DATA_BLOCK "NC"	// DB 10
VERSION : 0.0
  STRUCT
   A_Disabl_Inp1 : BOOL ;	//Disable digi. NCK input 1
   A_Disabl_Inp2 : BOOL ;	//Disable digi. NCK input 2
   A_Disabl_Inp3 : BOOL ;	//Disable digi. NCK input 3
   A_Disabl_Inp4 : BOOL ;	//Disable digi. NCK input 4
   A_Disabl_Inp5 : BOOL ;	//Disable digi. NCK input 5
   A_Disabl_Inp6 : BOOL ;	//Disable digi. NCK input 6
   A_Disabl_Inp7 : BOOL ;	//Disable digi. NCK input 7
   A_Disabl_Inp8 : BOOL ;	//Disable digi. NCK input 8
   A_Set_Inp1 : BOOL ;	//Set digi. NCK input 1
   A_Set_Inp2 : BOOL ;	//Set digi. NCK input 2
   A_Set_Inp3 : BOOL ;	//Set digi. NCK input 3
   A_Set_Inp4 : BOOL ;	//Set digi. NCK input 4
   A_Set_Inp5 : BOOL ;	//Set digi. NCK input 5
   A_Set_Inp6 : BOOL ;	//Set digi. NCK input 6
   A_Set_Inp7 : BOOL ;	//Set digi. NCK input 7
   A_Set_Inp8 : BOOL ;	//Set digi. NCK input 8
   f0_f15 : ARRAY  [0 .. 15 ] OF BOOL ;	//Reserved
   A_Disabl_Out1 : BOOL ;	//Disable digi. NCK output 1
   A_Disabl_Out2 : BOOL ;	//Disable digi. NCK output 2
   A_Disabl_Out3 : BOOL ;	//Disable digi. NCK output 3
   A_Disabl_Out4 : BOOL ;	//Disable digi. NCK output 4
   A_Disabl_Out5 : BOOL ;	//Disable digi. NCK output 5
   A_Disabl_Out6 : BOOL ;	//Disable digi. NCK output 6
   A_Disabl_Out7 : BOOL ;	//Disable digi. NCK output 7
   A_Disabl_Out8 : BOOL ;	//Disable digi. NCK output 8
   A_OvMask_Out1 : BOOL ;	//Overwrite mask of digi. output 1
   A_OvMask_Out2 : BOOL ;	//Overwrite mask of digi. output 2
   A_OvMask_Out3 : BOOL ;	//Overwrite mask of digi. output 3
   A_OvMask_Out4 : BOOL ;	//Overwrite mask of digi. output 4
   A_OvMask_Out5 : BOOL ;	//Overwrite mask of digi. output 5
   A_OvMask_Out6 : BOOL ;	//Overwrite mask of digi. output 6
   A_OvMask_Out7 : BOOL ;	//Overwrite mask of digi. output 7
   A_OvMask_Out8 : BOOL ;	//Overwrite mask of digi. output 8
   A_Set_Out1 : BOOL ;	//Set digi. NCK output 1
   A_Set_Out2 : BOOL ;	//Set digi. NCK output 2
   A_Set_Out3 : BOOL ;	//Set digi. NCK output 3
   A_Set_Out4 : BOOL ;	//Set digi. NCK output 4
   A_Set_Out5 : BOOL ;	//Set digi. NCK output 5
   A_Set_Out6 : BOOL ;	//Set digi. NCK output 6
   A_Set_Out7 : BOOL ;	//Set digi. NCK output 7
   A_Set_Out8 : BOOL ;	//Set digi. NCK output 8
   A_InMask_Out1 : BOOL ;	//Input mask of digi. output 1
   A_InMask_Out2 : BOOL ;	//Input mask of digi. output 2
   A_InMask_Out3 : BOOL ;	//Input mask of digi. output 3
   A_InMask_Out4 : BOOL ;	//Input mask of digi. output 4
   A_InMask_Out5 : BOOL ;	//Input mask of digi. output 5
   A_InMask_Out6 : BOOL ;	//Input mask of digi. output 6
   A_InMask_Out7 : BOOL ;	//Input mask of digi. output 7
   A_InMask_Out8 : BOOL ;	//Input mask of digi. output 8
   MCP1AxisTbl : ARRAY  [1 .. 22 ] OF BYTE  := B#16#1, B#16#2, B#16#3, B#16#4, B#16#5, B#16#6, B#16#7, B#16#8, B#16#9, B#16#A, B#16#B, B#16#C;	//Axis No. Table MCP1
   MCP1MaxAxis : WORD ;	//max. of Axisno, must be smaller or equal gp_par.MaxAxis
   MCP2AxisTbl : ARRAY  [1 .. 22 ] OF BYTE  := B#16#1, B#16#2, B#16#3, B#16#4, B#16#5, B#16#6, B#16#7, B#16#8, B#16#9, B#16#A, B#16#B, B#16#C;	//Axis No. Table MCP2
   MCP2MaxAxis : WORD ;	//max. of Axisno, must be smaller or equal gp_par.MaxAxis
   f56_0 : BOOL ;
   A_EMERGENCY : BOOL ;	//Emergency stop
   A_EMERGENCY_Ackn : BOOL ;	//Acknowledge emergency stop
   f56_3 : BOOL ;
   A_Keyswitch0 : BOOL ;	//Keyswitch position 0
   A_Keyswitch1 : BOOL ;	//Keyswitch position 1
   A_Keyswitch2 : BOOL ;	//Keyswitch position 2
   A_Keyswitch3 : BOOL ;	//Keyswitch position 3
   A_IncInModeGroup : BOOL ;	//INC inputs in mode group area active
   f57_1 : BOOL ;
   f57_2 : BOOL ;
   A_PCshutdown : BOOL ;	//PC shutdown 840Di
   f57_4 : BOOL ;
   f57_5 : BOOL ;
   f57_6 : BOOL ;
   f57_7 : BOOL ;
   A_CollCheckOff : BOOL ;	//Collisions Check Off
   f58_1 : BOOL ;
   f58_2 : BOOL ;
   f58_3 : BOOL ;
   f58_4 : BOOL ;
   f58_5 : BOOL ;
   f58_6 : BOOL ;
   f58_7 : BOOL ;
   f59 : BYTE ;
   E_ActVal_In1 : BOOL ;	//Actual value of digi. NCK input 1
   E_ActVal_In2 : BOOL ;	//Actual value of digi. NCK input 2
   E_ActVal_In3 : BOOL ;	//Actual value of digi. NCK input 3
   E_ActVal_In4 : BOOL ;	//Actual value of digi. NCK input 4
   f60_4 : BOOL ;
   f60_5 : BOOL ;
   f60_6 : BOOL ;
   f60_7 : BOOL ;
   f61_f62 : ARRAY  [61 .. 61 ] OF BYTE ;
   E_Setpoint_Out1 : BOOL ;	//Setpoint of digi. NCK output 1
   E_Setpoint_Out2 : BOOL ;	//Setpoint of digi. NCK output 2
   E_Setpoint_Out3 : BOOL ;	//Setpoint of digi. NCK output 3
   E_Setpoint_Out4 : BOOL ;	//Setpoint of digi. NCK output 4
   E_Setpoint_Out5 : BOOL ;	//Setpoint of digi. NCK output 5
   E_Setpoint_Out6 : BOOL ;	//Setpoint of digi. NCK output 6
   E_Setpoint_Out7 : BOOL ;	//Setpoint of digi. NCK output 7
   E_Setpoint_Out8 : BOOL ;	//Setpoint of digi. NCK output 8
   f65_f67 : ARRAY  [65 .. 66 ] OF BYTE ;
   E_HW1_moved : BYTE ;	//Handwheel 1 moved
   E_HW2_moved : BYTE ;	//Handwheel 2 moved
   E_HW3_moved : BYTE ;	//Handwheel 3 moved
   E_CounterInchMetr : BYTE ;	//Modification counter inch/metric system of units
   E_MCP1AxisValid : BOOL ;	//from HT6
   E_MCP1WCS : BOOL ;	//from HT6
   f72_2 : BOOL ;
   f72_3 : BOOL ;
   f72_4 : BOOL ;
   f72_5 : BOOL ;
   f72_6 : BOOL ;
   E_MCP1AxKeyDisp : BOOL ;	//Mcp1 Axis Key Displayed
   E_MCP2AxisValid : BOOL ;	//from HT6
   E_MCP2WCS : BOOL ;	//from HT6
   f73_2 : BOOL ;
   f73_3 : BOOL ;
   f73_4 : BOOL ;
   f73_5 : BOOL ;
   f73_6 : BOOL ;
   E_MCP2AxKeyDisp : BOOL ;	//Mcp2 Axis Key Displayed
   MCP1AxisFromHMI : ARRAY  [1 .. 6 ] OF BYTE ;	//Axistable from HT6
   MCP2AxisFromHMI : ARRAY  [1 .. 6 ] OF BYTE ;	//Axistable from HT6
   res86 : WORD ;
   res88 : BYTE ;
   res89 : BYTE ;
   epsToPlc : BYTE ;
   epsFromPlc : BYTE ;
   MpiDpOk : BOOL ;	//Slaves on MPI/DP Ok
   DpOk : BOOL ;	//Slaves on DP Ok
   f92_2 : BOOL ;
   f92_3 : BOOL ;
   f92_4 : BOOL ;
   f92_5 : BOOL ;
   f92_6 : BOOL ;
   f92_7 : BOOL ;
   f93 : BYTE ;
   f94 : BYTE ;
   f95 : BYTE ;
   E_LanguageID : BYTE ;	// LanguageID on HMI
   E_Chan_HW1_A : BOOL ;	//Channel number for handwheel1 A
   E_Chan_HW1_B : BOOL ;	//Channel number for handwheel1 B
   E_Chan_HW1_C : BOOL ;	//Channel number for handwheel1 C
   E_Chan_HW1_D : BOOL ;	//Channel number for handwheel1 D
   f97_4 : BOOL ;
   f97_5 : BOOL ;
   f97_6 : BOOL ;
   f97_7 : BOOL ;
   E_Chan_HW2_A : BOOL ;	//Channel number for handwheel2 A
   E_Chan_HW2_B : BOOL ;	//Channel number for handwheel2 B
   E_Chan_HW2_C : BOOL ;	//Channel number for handwheel2 C
   E_Chan_HW2_D : BOOL ;	//Channel number for handwheel2 D
   f98_4 : BOOL ;
   f98_5 : BOOL ;
   f98_6 : BOOL ;
   f98_7 : BOOL ;
   E_Chan_HW3_A : BOOL ;	//Channel number for handwheel3 A
   E_Chan_HW3_B : BOOL ;	//Channel number for handwheel3 B
   E_Chan_HW3_C : BOOL ;	//Channel number for handwheel3 C
   E_Chan_HW3_D : BOOL ;	//Channel number for handwheel3 D
   f99_4 : BOOL ;
   f99_5 : BOOL ;
   f99_6 : BOOL ;
   f99_7 : BOOL ;
   E_Ax_A_HW1 : BOOL ;	//Axis number for handwheel1 A
   E_Ax_B_HW1 : BOOL ;	//Axis number for handwheel1 B
   E_Ax_C_HW1 : BOOL ;	//Axis number for handwheel1 C
   E_Ax_D_HW1 : BOOL ;	//Axis number for handwheel1 D
   E_Ax_E_HW1 : BOOL ;	//Axis number for handwheel1 E
   E_CHW_sel1 : BOOL ;	//Contour handwheel selected
   E_HW_sel1 : BOOL ;	//Handwheel selected
   E_Mach_Ax1 : BOOL ;	//Machine axis
   E_Ax_A_HW2 : BOOL ;	//Axis number for handwheel2 A
   E_Ax_B_HW2 : BOOL ;	//Axis number for handwheel2 B
   E_Ax_C_HW2 : BOOL ;	//Axis number for handwheel2 C
   E_Ax_D_HW2 : BOOL ;	//Axis number for handwheel2 D
   E_Ax_E_HW2 : BOOL ;	//Axis number for handwheel2 E
   E_CHW_sel2 : BOOL ;	//Contour handwheel selected
   E_HW_sel2 : BOOL ;	//Handwheel selected
   E_Mach_Ax2 : BOOL ;	//Machine axis
   E_Ax_A_HW3 : BOOL ;	//Axis number for handwheel3 A
   E_Ax_B_HW3 : BOOL ;	//Axis number for handwheel3 B
   E_Ax_C_HW3 : BOOL ;	//Axis number for handwheel3 C
   E_Ax_D_HW3 : BOOL ;	//Axis number for handwheel3 D
   E_Ax_E_HW3 : BOOL ;	//Axis number for handwheel3 E
   E_CHW_sel3 : BOOL ;	//Contour handwheel selected
   E_HW_sel3 : BOOL ;	//Handwheel selected
   E_Mach_Ax3 : BOOL ;	//Machine axis
   E_RemDiag : BOOL ;	//Remote Diagnostic
   f103_1 : BOOL ;
   f103_2 : BOOL ;
   f103_3 : BOOL ;
   f103_4 : BOOL ;
   E_ATready : BOOL ;	//AT-box ready
   E_MMCTemp : BOOL ;	//MMC temperature limit
   E_MMCBatt : BOOL ;	//MMC 101/102 battery alarm
   E_MCP1ready : BOOL ;	//MCP1 ready;
   E_MCP2ready : BOOL ;	//MCP2 ready;
   E_BHGready : BOOL ;	//BHG ready;
   f104_3 : BOOL ;
   f104_4 : BOOL ;
   f104_5 : BOOL ;
   E_FirstOB1 : BOOL ;	//This bit is on for the first OB1 cycle
   E_NCKready : BOOL ;	//NCK CPU ready
   E_CancelToolCmd : BOOL ;	//Terminate canceled tool command
   f105_1 : BOOL ;
   f105_2 : BOOL ;
   f105_3 : BOOL ;
   f105_4 : BOOL ;
   f105_5 : BOOL ;
   f105_6 : BOOL ;
   f105_7 : BOOL ;
   E_CollCheckOff : BOOL ;	//CollisionsCheck Off
   E_EMSTOP : BOOL ;	//EMERGENCY STOP active
   f106_2 : BOOL ;
   f106_3 : BOOL ;
   f106_4 : BOOL ;
   f106_5 : BOOL ;
   f106_6 : BOOL ;
   f106_7 : BOOL ;
   E_InspProbe1 : BOOL ;	//Inspection probe 1 actuated
   E_InspProbe2 : BOOL ;	//Inspection probe 2 actuated
   f107_2 : BOOL ;
   f107_3 : BOOL ;
   f107_4 : BOOL ;
   f107_5 : BOOL ;
   E_NCU_LinkActive : BOOL ;	//NCU link active
   E_SystemInchDim : BOOL ;	//System inch dimension
   f108_0 : BOOL ;
   E_MMC2Ready : BOOL ;	//MMC2-CPU ready
   E_MMCMPIready : BOOL ;	//MMC1-CPU on MPI ready
   E_MMCBTSSready : BOOL ;	//MMC1-CPU on BTSS ready
   f108_4 : BOOL ;
   E_DrivesInCylOp : BOOL ;	//Drives in cylindric operation
   E_611Dready : BOOL ;	//611D ready
   E_NCready : BOOL ;
   E_NCKalarm : BOOL ;	//NCK alarm present
   f109_1 : BOOL ;
   f109_2 : BOOL ;
   f109_3 : BOOL ;
   A_PC_OSfault : BOOL ;	//PC operating system fault, 840Di
   E_HTempAlarm : BOOL ;	//Heat sink temperature alarm NCU 573
   E_ATempAlarm : BOOL ;	//Air temperature alarm
   E_BattAlarm : BOOL ;	//NCK battery alarm
   E_SWCamMinus : ARRAY  [0 .. 31 ] OF BOOL ;	//Software cams minus [0..31]
   E_SWCamPlus : ARRAY  [0 .. 31 ] OF BOOL ;	//Software cams plus [0..31]
   f118_f121 : ARRAY  [0 .. 3 ] OF BYTE ;
   A_Disabl_Inp9 : BOOL ;	//Disable digi. NCK input 9
   A_Disabl_Inp10 : BOOL ;	//Disable digi. NCK input 10
   A_Disabl_Inp11 : BOOL ;	//Disable digi. NCK input 11
   A_Disabl_Inp12 : BOOL ;	//Disable digi. NCK input 12
   A_Disabl_Inp13 : BOOL ;	//Disable digi. NCK input 13
   A_Disabl_Inp14 : BOOL ;	//Disable digi. NCK input 14
   A_Disabl_Inp15 : BOOL ;	//Disable digi. NCK input 15
   A_Disabl_Inp16 : BOOL ;	//Disable digi. NCK input 16
   A_Set_Inp9 : BOOL ;	//Set digi. NCK input 9
   A_Set_Inp10 : BOOL ;	//Set digi. NCK input 10
   A_Set_Inp11 : BOOL ;	//Set digi. NCK input 11
   A_Set_Inp12 : BOOL ;	//Set digi. NCK input 12
   A_Set_Inp13 : BOOL ;	//Set digi. NCK input 13
   A_Set_Inp14 : BOOL ;	//Set digi. NCK input 14
   A_Set_Inp15 : BOOL ;	//Set digi. NCK input 15
   A_Set_Inp16 : BOOL ;	//Set digi. NCK input 16
   A_Disabl_Inp17 : BOOL ;	//Disable digi. NCK input 17
   A_Disabl_Inp18 : BOOL ;	//Disable digi. NCK input 18
   A_Disabl_Inp19 : BOOL ;	//Disable digi. NCK input 19
   A_Disabl_Inp20 : BOOL ;	//Disable digi. NCK input 20
   A_Disabl_Inp21 : BOOL ;	//Disable digi. NCK input 21
   A_Disabl_Inp22 : BOOL ;	//Disable digi. NCK input 22
   A_Disabl_Inp23 : BOOL ;	//Disable digi. NCK input 23
   A_Disabl_Inp24 : BOOL ;	//Disable digi. NCK input 24
   A_Set_Inp17 : BOOL ;	//Set digi. NCK input 17
   A_Set_Inp18 : BOOL ;	//Set digi. NCK input 18
   A_Set_Inp19 : BOOL ;	//Set digi. NCK input 19
   A_Set_Inp20 : BOOL ;	//Set digi. NCK input 20
   A_Set_Inp21 : BOOL ;	//Set digi. NCK input 21
   A_Set_Inp22 : BOOL ;	//Set digi. NCK input 22
   A_Set_Inp23 : BOOL ;	//Set digi. NCK input 23
   A_Set_Inp24 : BOOL ;	//Set digi. NCK input 24
   A_Disabl_Inp25 : BOOL ;	//Disable digi. NCK input 25
   A_Disabl_Inp26 : BOOL ;	//Disable digi. NCK input 26
   A_Disabl_Inp27 : BOOL ;	//Disable digi. NCK input 27
   A_Disabl_Inp28 : BOOL ;	//Disable digi. NCK input 28
   A_Disabl_Inp29 : BOOL ;	//Disable digi. NCK input 29
   A_Disabl_Inp30 : BOOL ;	//Disable digi. NCK input 30
   A_Disabl_Inp31 : BOOL ;	//Disable digi. NCK input 31
   A_Disabl_Inp32 : BOOL ;	//Disable digi. NCK input 32
   A_Set_Inp25 : BOOL ;	//Set digi. NCK input 25
   A_Set_Inp26 : BOOL ;	//Set digi. NCK input 26
   A_Set_Inp27 : BOOL ;	//Set digi. NCK input 27
   A_Set_Inp28 : BOOL ;	//Set digi. NCK input 28
   A_Set_Inp29 : BOOL ;	//Set digi. NCK input 29
   A_Set_Inp30 : BOOL ;	//Set digi. NCK input 30
   A_Set_Inp31 : BOOL ;	//Set digi. NCK input 31
   A_Set_Inp32 : BOOL ;	//Set digi. NCK input 32
   A_Disabl_Inp33 : BOOL ;	//Disable digi. NCK input 33
   A_Disabl_Inp34 : BOOL ;	//Disable digi. NCK input 34
   A_Disabl_Inp35 : BOOL ;	//Disable digi. NCK input 35
   A_Disabl_Inp36 : BOOL ;	//Disable digi. NCK input 36
   A_Disabl_Inp37 : BOOL ;	//Disable digi. NCK input 37
   A_Disabl_Inp38 : BOOL ;	//Disable digi. NCK input 38
   A_Disabl_Inp39 : BOOL ;	//Disable digi. NCK input 39
   A_Disabl_Inp40 : BOOL ;	//Disable digi. NCK input 40
   A_Set_Inp33 : BOOL ;	//Set digi. NCK input 33
   A_Set_Inp34 : BOOL ;	//Set digi. NCK input 34
   A_Set_Inp35 : BOOL ;	//Set digi. NCK input 35
   A_Set_Inp36 : BOOL ;	//Set digi. NCK input 36
   A_Set_Inp37 : BOOL ;	//Set digi. NCK input 37
   A_Set_Inp38 : BOOL ;	//Set digi. NCK input 38
   A_Set_Inp39 : BOOL ;	//Set digi. NCK input 39
   A_Set_Inp40 : BOOL ;	//Set digi. NCK input 40
   A_Disabl_Out9 : BOOL ;	//Disable digi. NCK output 9
   A_Disabl_Out10 : BOOL ;	//Disable digi. NCK output 10
   A_Disabl_Out11 : BOOL ;	//Disable digi. NCK output 11
   A_Disabl_Out12 : BOOL ;	//Disable digi. NCK output 12
   A_Disabl_Out13 : BOOL ;	//Disable digi. NCK output 13
   A_Disabl_Out14 : BOOL ;	//Disable digi. NCK output 14
   A_Disabl_Out15 : BOOL ;	//Disable digi. NCK output 15
   A_Disabl_Out16 : BOOL ;	//Disable digi. NCK output 16
   A_OvMask_Out9 : BOOL ;	//Overwrite mask of digi. output 9
   A_OvMask_Out10 : BOOL ;	//Overwrite mask of digi. output 10
   A_OvMask_Out11 : BOOL ;	//Overwrite mask of digi. output 11
   A_OvMask_Out12 : BOOL ;	//Overwrite mask of digi. output 12
   A_OvMask_Out13 : BOOL ;	//Overwrite mask of digi. output 13
   A_OvMask_Out14 : BOOL ;	//Overwrite mask of digi. output 14
   A_OvMask_Out15 : BOOL ;	//Overwrite mask of digi. output 15
   A_OvMask_Out16 : BOOL ;	//Overwrite mask of digi. output 16
   A_Setval_Out9 : BOOL ;	//Set value digi. NCK output 9
   A_Setval_Out10 : BOOL ;	//Set value digi. NCK output 10
   A_Setval_Out11 : BOOL ;	//Set value digi. NCK output 11
   A_Setval_Out12 : BOOL ;	//Set value digi. NCK output 12
   A_Setval_Out13 : BOOL ;	//Set value digi. NCK output 13
   A_Setval_Out14 : BOOL ;	//Set value digi. NCK output 14
   A_Setval_Out15 : BOOL ;	//Set value digi. NCK output 15
   A_Setval_Out16 : BOOL ;	//Set value digi. NCK output 16
   A_InMask_Out9 : BOOL ;	//Input mask of digi. output 9
   A_InMask_Out10 : BOOL ;	//Input mask of digi. output 10
   A_InMask_Out11 : BOOL ;	//Input mask of digi. output 11
   A_InMask_Out12 : BOOL ;	//Input mask of digi. output 12
   A_InMask_Out13 : BOOL ;	//Input mask of digi. output 13
   A_InMask_Out14 : BOOL ;	//Input mask of digi. output 14
   A_InMask_Out15 : BOOL ;	//Input mask of digi. output 15
   A_InMask_Out16 : BOOL ;	//Input mask of digi. output 16
   A_Disabl_Out17 : BOOL ;	//Disable digi. NCK output 17
   A_Disabl_Out18 : BOOL ;	//Disable digi. NCK output 18
   A_Disabl_Out19 : BOOL ;	//Disable digi. NCK output 19
   A_Disabl_Out20 : BOOL ;	//Disable digi. NCK output 20
   A_Disabl_Out21 : BOOL ;	//Disable digi. NCK output 21
   A_Disabl_Out22 : BOOL ;	//Disable digi. NCK output 22
   A_Disabl_Out23 : BOOL ;	//Disable digi. NCK output 23
   A_Disabl_Out24 : BOOL ;	//Disable digi. NCK output 24
   A_OvMask_Out17 : BOOL ;	//Overwrite mask of digi. output 17
   A_OvMask_Out18 : BOOL ;	//Overwrite mask of digi. output 18
   A_OvMask_Out19 : BOOL ;	//Overwrite mask of digi. output 19
   A_OvMask_Out20 : BOOL ;	//Overwrite mask of digi. output 20
   A_OvMask_Out21 : BOOL ;	//Overwrite mask of digi. output 21
   A_OvMask_Out22 : BOOL ;	//Overwrite mask of digi. output 22
   A_OvMask_Out23 : BOOL ;	//Overwrite mask of digi. output 23
   A_OvMask_Out24 : BOOL ;	//Overwrite mask of digi. output 24
   A_Setval_Out17 : BOOL ;	//Set value digi. NCK output 17
   A_Setval_Out18 : BOOL ;	//Set value digi. NCK output 18
   A_Setval_Out19 : BOOL ;	//Set value digi. NCK output 19
   A_Setval_Out20 : BOOL ;	//Set value digi. NCK output 20
   A_Setval_Out21 : BOOL ;	//Set value digi. NCK output 21
   A_Setval_Out22 : BOOL ;	//Set value digi. NCK output 22
   A_Setval_Out23 : BOOL ;	//Set value digi. NCK output 23
   A_Setval_Out24 : BOOL ;	//Set value digi. NCK output 24
   A_InMask_Out17 : BOOL ;	//Input mask of digi. output 17
   A_InMask_Out18 : BOOL ;	//Input mask of digi. output 18
   A_InMask_Out19 : BOOL ;	//Input mask of digi. output 19
   A_InMask_Out20 : BOOL ;	//Input mask of digi. output 20
   A_InMask_Out21 : BOOL ;	//Input mask of digi. output 21
   A_InMask_Out22 : BOOL ;	//Input mask of digi. output 22
   A_InMask_Out23 : BOOL ;	//Input mask of digi. output 23
   A_InMask_Out24 : BOOL ;	//Input mask of digi. output 24
   A_Disabl_Out25 : BOOL ;	//Disable digi. NCK output 25
   A_Disabl_Out26 : BOOL ;	//Disable digi. NCK output 26
   A_Disabl_Out27 : BOOL ;	//Disable digi. NCK output 27
   A_Disabl_Out28 : BOOL ;	//Disable digi. NCK output 28
   A_Disabl_Out29 : BOOL ;	//Disable digi. NCK output 29
   A_Disabl_Out30 : BOOL ;	//Disable digi. NCK output 30
   A_Disabl_Out31 : BOOL ;	//Disable digi. NCK output 31
   A_Disabl_Out32 : BOOL ;	//Disable digi. NCK output 32
   A_OvMask_Out25 : BOOL ;	//Overwrite mask of digi. output 25
   A_OvMask_Out26 : BOOL ;	//Overwrite mask of digi. output 26
   A_OvMask_Out27 : BOOL ;	//Overwrite mask of digi. output 27
   A_OvMask_Out28 : BOOL ;	//Overwrite mask of digi. output 28
   A_OvMask_Out29 : BOOL ;	//Overwrite mask of digi. output 29
   A_OvMask_Out30 : BOOL ;	//Overwrite mask of digi. output 30
   A_OvMask_Out31 : BOOL ;	//Overwrite mask of digi. output 31
   A_OvMask_Out32 : BOOL ;	//Overwrite mask of digi. output 32
   A_Setval_Out25 : BOOL ;	//Set value digi. NCK output 25
   A_Setval_Out26 : BOOL ;	//Set value digi. NCK output 26
   A_Setval_Out27 : BOOL ;	//Set value digi. NCK output 27
   A_Setval_Out28 : BOOL ;	//Set value digi. NCK output 28
   A_Setval_Out29 : BOOL ;	//Set value digi. NCK output 29
   A_Setval_Out30 : BOOL ;	//Set value digi. NCK output 30
   A_Setval_Out31 : BOOL ;	//Set value digi. NCK output 31
   A_Setval_Out32 : BOOL ;	//Set value digi. NCK output 32
   A_InMask_Out25 : BOOL ;	//Input mask of digi. output 25
   A_InMask_Out26 : BOOL ;	//Input mask of digi. output 26
   A_InMask_Out27 : BOOL ;	//Input mask of digi. output 27
   A_InMask_Out28 : BOOL ;	//Input mask of digi. output 28
   A_InMask_Out29 : BOOL ;	//Input mask of digi. output 29
   A_InMask_Out30 : BOOL ;	//Input mask of digi. output 30
   A_InMask_Out31 : BOOL ;	//Input mask of digi. output 31
   A_InMask_Out32 : BOOL ;	//Input mask of digi. output 32
   A_Disabl_Out33 : BOOL ;	//Disable digi. NCK output 33
   A_Disabl_Out34 : BOOL ;	//Disable digi. NCK output 34
   A_Disabl_Out35 : BOOL ;	//Disable digi. NCK output 35
   A_Disabl_Out36 : BOOL ;	//Disable digi. NCK output 36
   A_Disabl_Out37 : BOOL ;	//Disable digi. NCK output 37
   A_Disabl_Out38 : BOOL ;	//Disable digi. NCK output 38
   A_Disabl_Out39 : BOOL ;	//Disable digi. NCK output 39
   A_Disabl_Out40 : BOOL ;	//Disable digi. NCK output 40
   A_OvMask_Out33 : BOOL ;	//Overwrite mask of digi. output 33
   A_OvMask_Out34 : BOOL ;	//Overwrite mask of digi. output 34
   A_OvMask_Out35 : BOOL ;	//Overwrite mask of digi. output 35
   A_OvMask_Out36 : BOOL ;	//Overwrite mask of digi. output 36
   A_OvMask_Out37 : BOOL ;	//Overwrite mask of digi. output 37
   A_OvMask_Out38 : BOOL ;	//Overwrite mask of digi. output 38
   A_OvMask_Out39 : BOOL ;	//Overwrite mask of digi. output 39
   A_OvMask_Out40 : BOOL ;	//Overwrite mask of digi. output 40
   A_Setval_out33 : BOOL ;	//Set value digi. NCK output 33
   A_Setval_out34 : BOOL ;	//Set value digi. NCK output 34
   A_Setval_out35 : BOOL ;	//Set value digi. NCK output 35
   A_Setval_out36 : BOOL ;	//Set value digi. NCK output 36
   A_Setval_out37 : BOOL ;	//Set value digi. NCK output 37
   A_Setval_out38 : BOOL ;	//Set value digi. NCK output 38
   A_Setval_out39 : BOOL ;	//Set value digi. NCK output 39
   A_Setval_out40 : BOOL ;	//Set value digi. NCK output 40
   A_InMask_Out33 : BOOL ;	//Input mask of digi. output 33
   A_InMask_Out34 : BOOL ;	//Input mask of digi. output 34
   A_InMask_Out35 : BOOL ;	//Input mask of digi. output 35
   A_InMask_Out36 : BOOL ;	//Input mask of digi. output 36
   A_InMask_Out37 : BOOL ;	//Input mask of digi. output 37
   A_InMask_Out38 : BOOL ;	//Input mask of digi. output 38
   A_InMask_Out39 : BOOL ;	//Input mask of digi. output 39
   A_InMask_Out40 : BOOL ;	//Input mask of digi. output 40
   A_Disabl_anaIn1 : BOOL ;	//Disable analog NCK input 1
   A_Disabl_anaIn2 : BOOL ;	//Disable analog NCK input 2
   A_Disabl_anaIn3 : BOOL ;	//Disable analog NCK input 3
   A_Disabl_anaIn4 : BOOL ;	//Disable analog NCK input 4
   A_Disabl_anaIn5 : BOOL ;	//Disable analog NCK input 5
   A_Disabl_anaIn6 : BOOL ;	//Disable analog NCK input 6
   A_Disabl_anaIn7 : BOOL ;	//Disable analog NCK input 7
   A_Disabl_anaIn8 : BOOL ;	//Disable analog NCK input 8
   A_InMask_anaIn1 : BOOL ;	//Input mask of analog NCK input 1
   A_InMask_anaIn2 : BOOL ;	//Input mask of analog NCK input 2
   A_InMask_anaIn3 : BOOL ;	//Input mask of analog NCK input 3
   A_InMask_anaIn4 : BOOL ;	//Input mask of analog NCK input 4
   A_InMask_anaIn5 : BOOL ;	//Input mask of analog NCK input 5
   A_InMask_anaIn6 : BOOL ;	//Input mask of analog NCK input 6
   A_InMask_anaIn7 : BOOL ;	//Input mask of analog NCK input 7
   A_InMask_anaIn8 : BOOL ;	//Input mask of analog NCK input 8
   A_Setval_anaIn1 : WORD ;	//Set value of analog NCK input 1
   A_Setval_anaIn2 : WORD ;	//Set value of analog NCK input 2
   A_Setval_anaIn3 : WORD ;	//Set value of analog NCK input 3
   A_Setval_anaIn4 : WORD ;	//Set value of analog NCK input 4
   A_Setval_anaIn5 : WORD ;	//Set value of analog NCK input 5
   A_Setval_anaIn6 : WORD ;	//Set value of analog NCK input 6
   A_Setval_anaIn7 : WORD ;	//Set value of analog NCK input 7
   A_Setval_anaIn8 : WORD ;	//Set value of analog NCK input 8
   f164_f165 : INT ;
   A_OvMask_anaOut1 : BOOL ;	//Overwrite mask of analog output 1
   A_OvMask_anaOut2 : BOOL ;	//Overwrite mask of analog output 2
   A_OvMask_anaOut3 : BOOL ;	//Overwrite mask of analog output 3
   A_OvMask_anaOut4 : BOOL ;	//Overwrite mask of analog output 4
   A_OvMask_anaOut5 : BOOL ;	//Overwrite mask of analog output 5
   A_OvMask_anaOut6 : BOOL ;	//Overwrite mask of analog output 6
   A_OvMask_anaOut7 : BOOL ;	//Overwrite mask of analog output 7
   A_OvMask_anaOut8 : BOOL ;	//Overwrite mask of analog output 8
   A_InMask_anaOut1 : BOOL ;	//Input mask of analog NCK output 1
   A_InMask_anaOut2 : BOOL ;	//Input mask of analog NCK output 2
   A_InMask_anaOut3 : BOOL ;	//Input mask of analog NCK output 3
   A_InMask_anaOut4 : BOOL ;	//Input mask of analog NCK output 4
   A_InMask_anaOut5 : BOOL ;	//Input mask of analog NCK output 5
   A_InMask_anaOut6 : BOOL ;	//Input mask of analog NCK output 6
   A_InMask_anaOut7 : BOOL ;	//Input mask of analog NCK output 7
   A_InMask_anaOut8 : BOOL ;	//Input mask of analog NCK output 8
   A_Disabl_anaOut1 : BOOL ;	//Disable analog NCK output 1
   A_Disabl_anaOut2 : BOOL ;	//Disable analog NCK output 2
   A_Disabl_anaOut3 : BOOL ;	//Disable analog NCK output 3
   A_Disabl_anaOut4 : BOOL ;	//Disable analog NCK output 4
   A_Disabl_anaOut5 : BOOL ;	//Disable analog NCK output 5
   A_Disabl_anaOut6 : BOOL ;	//Disable analog NCK output 6
   A_Disabl_anaOut7 : BOOL ;	//Disable analog NCK output 7
   A_Disabl_anaOut8 : BOOL ;	//Disable analog NCK output 8
   f169 : BYTE ;
   A_Setval_anaOut1 : WORD ;	//Set value of analog NCK output 1
   A_Setval_anaOut2 : WORD ;	//Set value of analog NCK output 2
   A_Setval_anaOut3 : WORD ;	//Set value of analog NCK output 3
   A_Setval_anaOut4 : WORD ;	//Set value of analog NCK output 4
   A_Setval_anaOut5 : WORD ;	//Set value of analog NCK output 5
   A_Setval_anaOut6 : WORD ;	//Set value of analog NCK output 6
   A_Setval_anaOut7 : WORD ;	//Set value of analog NCK output 7
   A_Setval_anaOut8 : WORD ;	//Set value of analog NCK output 8
   E_ActVal_In9 : BOOL ;	//Actual value of digi. NCK input 9
   E_ActVal_In10 : BOOL ;	//Actual value of digi. NCK input 10
   E_ActVal_In11 : BOOL ;	//Actual value of digi. NCK input 11
   E_ActVal_In12 : BOOL ;	//Actual value of digi. NCK input 12
   E_ActVal_In13 : BOOL ;	//Actual value of digi. NCK input 13
   E_ActVal_In14 : BOOL ;	//Actual value of digi. NCK input 14
   E_ActVal_In15 : BOOL ;	//Actual value of digi. NCK input 15
   E_ActVal_In16 : BOOL ;	//Actual value of digi. NCK input 16
   E_ActVal_In17 : BOOL ;	//Actual value of digi. NCK input 17
   E_ActVal_In18 : BOOL ;	//Actual value of digi. NCK input 18
   E_ActVal_In19 : BOOL ;	//Actual value of digi. NCK input 19
   E_ActVal_In20 : BOOL ;	//Actual value of digi. NCK input 20
   E_ActVal_In21 : BOOL ;	//Actual value of digi. NCK input 21
   E_ActVal_In22 : BOOL ;	//Actual value of digi. NCK input 22
   E_ActVal_In23 : BOOL ;	//Actual value of digi. NCK input 23
   E_ActVal_In24 : BOOL ;	//Actual value of digi. NCK input 24
   E_ActVal_In25 : BOOL ;	//Actual value of digi. NCK input 25
   E_ActVal_In26 : BOOL ;	//Actual value of digi. NCK input 26
   E_ActVal_In27 : BOOL ;	//Actual value of digi. NCK input 27
   E_ActVal_In28 : BOOL ;	//Actual value of digi. NCK input 28
   E_ActVal_In29 : BOOL ;	//Actual value of digi. NCK input 29
   E_ActVal_In30 : BOOL ;	//Actual value of digi. NCK input 30
   E_ActVal_In31 : BOOL ;	//Actual value of digi. NCK input 31
   E_ActVal_In32 : BOOL ;	//Actual value of digi. NCK input 32
   E_ActVal_In33 : BOOL ;	//Actual value of digi. NCK input 33
   E_ActVal_In34 : BOOL ;	//Actual value of digi. NCK input 34
   E_ActVal_In35 : BOOL ;	//Actual value of digi. NCK input 35
   E_ActVal_In36 : BOOL ;	//Actual value of digi. NCK input 36
   E_ActVal_In37 : BOOL ;	//Actual value of digi. NCK input 37
   E_ActVal_In38 : BOOL ;	//Actual value of digi. NCK input 38
   E_ActVal_In39 : BOOL ;	//Actual value of digi. NCK input 39
   E_ActVal_In40 : BOOL ;	//Actual value of digi. NCK input 40
   E_Setpoint_Out9 : BOOL ;	//Setpoint of digi. NCK output 9
   E_Setpoint_Out10 : BOOL ;	//Setpoint of digi. NCK output 10
   E_Setpoint_Out11 : BOOL ;	//Setpoint of digi. NCK output 11
   E_Setpoint_Out12 : BOOL ;	//Setpoint of digi. NCK output 12
   E_Setpoint_Out13 : BOOL ;	//Setpoint of digi. NCK output 13
   E_Setpoint_Out14 : BOOL ;	//Setpoint of digi. NCK output 14
   E_Setpoint_Out15 : BOOL ;	//Setpoint of digi. NCK output 15
   E_Setpoint_Out16 : BOOL ;	//Setpoint of digi. NCK output 16
   E_Setpoint_Out17 : BOOL ;	//Setpoint of digi. NCK output 17
   E_Setpoint_Out18 : BOOL ;	//Setpoint of digi. NCK output 18
   E_Setpoint_Out19 : BOOL ;	//Setpoint of digi. NCK output 19
   E_Setpoint_Out20 : BOOL ;	//Setpoint of digi. NCK output 20
   E_Setpoint_Out21 : BOOL ;	//Setpoint of digi. NCK output 21
   E_Setpoint_Out22 : BOOL ;	//Setpoint of digi. NCK output 22
   E_Setpoint_Out23 : BOOL ;	//Setpoint of digi. NCK output 23
   E_Setpoint_Out24 : BOOL ;	//Setpoint of digi. NCK output 24
   E_Setpoint_Out25 : BOOL ;	//Setpoint of digi. NCK output 25
   E_Setpoint_Out26 : BOOL ;	//Setpoint of digi. NCK output 26
   E_Setpoint_Out27 : BOOL ;	//Setpoint of digi. NCK output 27
   E_Setpoint_Out28 : BOOL ;	//Setpoint of digi. NCK output 28
   E_Setpoint_Out29 : BOOL ;	//Setpoint of digi. NCK output 29
   E_Setpoint_Out30 : BOOL ;	//Setpoint of digi. NCK output 30
   E_Setpoint_Out31 : BOOL ;	//Setpoint of digi. NCK output 31
   E_Setpoint_Out32 : BOOL ;	//Setpoint of digi. NCK output 32
   E_Setpoint_Out33 : BOOL ;	//Setpoint of digi. NCK output 33
   E_Setpoint_Out34 : BOOL ;	//Setpoint of digi. NCK output 34
   E_Setpoint_Out35 : BOOL ;	//Setpoint of digi. NCK output 35
   E_Setpoint_Out36 : BOOL ;	//Setpoint of digi. NCK output 36
   E_Setpoint_Out37 : BOOL ;	//Setpoint of digi. NCK output 37
   E_Setpoint_Out38 : BOOL ;	//Setpoint of digi. NCK output 38
   E_Setpoint_Out39 : BOOL ;	//Setpoint of digi. NCK output 39
   E_Setpoint_Out40 : BOOL ;	//Setpoint of digi. NCK output 40
   E_ActVal_anaIn1 : WORD ;	//Actual value of analog NCK input 1
   E_ActVal_anaIn2 : WORD ;	//Actual value of analog NCK input 2
   E_ActVal_anaIn3 : WORD ;	//Actual value of analog NCK input 3
   E_ActVal_anaIn4 : WORD ;	//Actual value of analog NCK input 4
   E_ActVal_anaIn5 : WORD ;	//Actual value of analog NCK input 5
   E_ActVal_anaIn6 : WORD ;	//Actual value of analog NCK input 6
   E_ActVal_anaIn7 : WORD ;	//Actual value of analog NCK input 7
   E_ActVal_anaIn8 : WORD ;	//Actual value of analog NCK input 8
   E_SetVal_anaOut1 : WORD ;	//Set value of analog NCK output 1
   E_SetVal_anaOut2 : WORD ;	//Set value of analog NCK output 2
   E_SetVal_anaOut3 : WORD ;	//Set value of analog NCK output 3
   E_SetVal_anaOut4 : WORD ;	//Set value of analog NCK output 4
   E_SetVal_anaOut5 : WORD ;	//Set value of analog NCK output 5
   E_SetVal_anaOut6 : WORD ;	//Set value of analog NCK output 6
   E_SetVal_anaOut7 : WORD ;	//Set value of analog NCK output 7
   E_SetVal_anaOut8 : WORD ;	//Set value of analog NCK output 8
   E_CollCheck : ARRAY  [0 .. 7 ] OF BYTE ;	//CollisionsCheck
   A_CollCheck : ARRAY  [0 .. 7 ] OF BYTE ;	//CollisionsCheck
   E_HW4_moved : BYTE ;	//Handwheel 4 moved
   E_HW5_moved : BYTE ;	//Handwheel 5 moved
   E_HW6_moved : BYTE ;	//Handwheel 6 moved
   E_EHW1_stands : BOOL ;	//Ethernet handwheel 1 stands
   E_EHW2_stands : BOOL ;	//Ethernet handwheel 2 stands
   E_EHW3_stands : BOOL ;	//Ethernet handwheel 3 stands
   E_EHW4_stands : BOOL ;	//Ethernet handwheel 4 stands
   E_EHW5_stands : BOOL ;	//Ethernet handwheel 5 stands
   E_EHW6_stands : BOOL ;	//Ethernet handwheel 6 stands
   f245_6 : BOOL ;
   f245_7 : BOOL ;
   f246 : WORD ;
  END_STRUCT ;	
BEGIN
   MCP1AxisTbl[1] := B#16#1;
   MCP1AxisTbl[2] := B#16#2;
   MCP1AxisTbl[3] := B#16#3;
   MCP1AxisTbl[4] := B#16#4;
   MCP1AxisTbl[5] := B#16#5;
   MCP1AxisTbl[6] := B#16#6;
   MCP1AxisTbl[7] := B#16#7;
   MCP1AxisTbl[8] := B#16#8;
   MCP1AxisTbl[9] := B#16#9;
   MCP1AxisTbl[10] := B#16#A;
   MCP1AxisTbl[11] := B#16#B;
   MCP1AxisTbl[12] := B#16#C;
   MCP2AxisTbl[1] := B#16#1;
   MCP2AxisTbl[2] := B#16#2;
   MCP2AxisTbl[3] := B#16#3;
   MCP2AxisTbl[4] := B#16#4;
   MCP2AxisTbl[5] := B#16#5;
   MCP2AxisTbl[6] := B#16#6;
   MCP2AxisTbl[7] := B#16#7;
   MCP2AxisTbl[8] := B#16#8;
   MCP2AxisTbl[9] := B#16#9;
   MCP2AxisTbl[10] := B#16#A;
   MCP2AxisTbl[11] := B#16#B;
   MCP2AxisTbl[12] := B#16#C;
END_DATA_BLOCK

DATA_BLOCK DB 15
AUTHOR : NUMERIK
FAMILY : _800D
NAME : Bas_Com
VERSION : 2.7
  STRUCT
   fifoFull : BOOL ;
   readOffset : BYTE ;
   writeOffset : BYTE ;
   filler : BYTE ;
   Fifo : ARRAY  [1 .. 10 ] OF BYTE ;
   pduRefArr : ARRAY  [1 .. 12 ] OF //Little Endian Werte
   STRUCT
    diNo : WORD ;
    diPartLen : WORD ;
    PdiBeg : DWORD ;
   END_STRUCT ;
  END_STRUCT ;	
BEGIN
END_DATA_BLOCK

// DB 16: know-how protected block, not included

DATA_BLOCK "SPL"	// DB 18
TITLE = SPL dataarea
AUTHOR : NUMERIK
FAMILY : _800D
NAME : Basics
VERSION : 2.7
  STRUCT
   INSEP_VALID : ARRAY  [1 .. 8 ] OF BOOL ;	//used external SPL-Inputbytes(HW)
   OUTSEP_VALID : ARRAY  [1 .. 8 ] OF BOOL ;	//used external SPL-Outputbytes(HW)
   INSEP_ADDR : ARRAY  [1 .. 8 ] OF INT ;	//Addresses external SPL-Inputbytes(HW)
   OUTSEP_ADDR : ARRAY  [1 .. 8 ] OF INT ;	//Addresses external SPL-Outputbytes(HW)
   SPL_READY : BOOL ;	//setup finished
   STOP_MODE : BOOL ;	//0= Stop D, 1=Stop E
   SPL_DATA : STRUCT
    INSEP : ARRAY  [1 .. 64 ] OF BOOL ;
    OUTSEP : ARRAY  [1 .. 64 ] OF BOOL ;
    INSIP : ARRAY  [1 .. 64 ] OF BOOL ;
    OUTSIP : ARRAY  [1 .. 64 ] OF BOOL ;
    MARKERSIP : ARRAY  [1 .. 64 ] OF BOOL ;
   END_STRUCT ;
   SPL_DELTA : STRUCT 	//edge difference NCK - PLC for Diagnostic
    INSEP : ARRAY  [1 .. 64 ] OF BOOL ;
    OUTSEP : ARRAY  [1 .. 64 ] OF BOOL ;
    INSIP : ARRAY  [1 .. 64 ] OF BOOL ;
    OUTSIP : ARRAY  [1 .. 64 ] OF BOOL ;
    MARKERSIP : ARRAY  [1 .. 64 ] OF BOOL ;
   END_STRUCT ;
   CMDSI : BOOL ;	//multiplication of Timeout Value by Factor 10
   CMDSI_R1 : BOOL ;	//for future use
   CMDSI_R2 : BOOL ;	//for future use
   CMDSI_R3 : BOOL ;	//for future use
   CMDSI_R4 : BOOL ;	//for future use
   CMDSI_R5 : BOOL ;	//for future use
   CMDSI_R6 : BOOL ;	//for future use
   CMDSI_R7 : BOOL ;	//for future use
   STATUS_R0 : BOOL ;	//for future use
   STATUS_R1 : BOOL ;	//for future use
   STATUS_R2 : BOOL ;	//for future use
   STATUS_R3 : BOOL ;	//for future use
   STATUS_R4 : BOOL ;	//for future use
   COMM_TO : BOOL ;	//Communication Timeout
   STATUS_R6 : BOOL ;	//for future use
   STATUS_R7 : BOOL ;	//for future use
   STATSI : DINT ;	//Status: 0 - no error, 1 - 320 error number
   LEVELSI : DINT ;	//stacklevel SPL-KDV for Diagnostic
   PLCSIOUT : ARRAY  [1 .. 32 ] OF BOOL ;	//Single Channel Signals from NCK
   PLCSIIN : ARRAY  [1 .. 32 ] OF BOOL ;	//Single Channel Signals to NCK
   SPL_STATUS : ARRAY  [1 .. 16 ] OF BOOL ;	//SPL Status from NCK
   INSEP_PROFISAFE : ARRAY  [1 .. 8 ] OF BOOL ;	//external SPL-Inputbytes(HW) with PROFIsafe Slaves
   OUTSEP_PROFISAFE : ARRAY  [1 .. 8 ] OF BOOL ;	//external SPL-Outputbytes(HW) with PROFIsafe Slaves
   NoOfAxisPerBlock : ARRAY  [1 .. 8 ] OF BYTE ;	//Pointer and Tables for Teststop
   BlockPointer : ARRAY  [1 .. 8 ] OF BYTE ;
   AxisTable : ARRAY  [1 .. 31 ] OF BYTE ;
   FSDP : ARRAY  [1 .. 3 ] OF STRUCT
    ERR_REAC : INT ;	// IN: Error reaction
    ERROR : BOOL ;	// OUT: 1=Communication error
    SUBS_ON : BOOL ;	// OUT: 1=Receiver outputs fail-safe values
    DIAG : WORD ;	// OUT: Service information
    RETVAL14 : WORD ;	// OUT: Error code of SFC 14
    RETVAL15 : WORD ;	// OUT: Error code of SFC 15
   END_STRUCT ;
   FRDP : ARRAY  [1 .. 3 ] OF STRUCT
    SUBS : ARRAY  [0 .. 15 ] OF BOOL ;	// IN: Fail-safe value for receive data BOOL 00 ... BOOL 15
    ERR_REAC : INT ;	// IN: Error reaction
    ACK_REI : BOOL ;	// IN: 1=Acknowledgment for reintegration of send data following communication er
    RES1 : BOOL ;	//Reserved
    RES2 : BOOL ;	//Reserved
    RES3 : BOOL ;	//Reserved
    RES4 : BOOL ;	//Reserved
    RES5 : BOOL ;	//Reserved
    RES6 : BOOL ;	//Reserved
    RES7 : BOOL ;	//Reserved
    ERROR : BOOL ;	// OUT: 1=Communication error
    SUBS_ON : BOOL ;	// OUT: 1=Fail-safe values are output
    ACK_REQ : BOOL ;	// OUT: 1=Acknowledgment for reintegration of send data required
    SENDMODE : BOOL ;	// OUT: 1=F_CPU with F_SENDDP in deactivated safety mode
    DIAG : WORD ;	// OUT: Service information
    RETVAL14 : WORD ;	// OUT: Error code of SFC 14
    RETVAL15 : WORD ;	// OUT: Error code of SFC 15
   END_STRUCT ;
   SPL_USER_DATA : ARRAY  [0 .. 3 ] OF DWORD ;
  END_STRUCT ;	
BEGIN
END_DATA_BLOCK

DATA_BLOCK "MMC"	// DB 19
VERSION : 0.0
  STRUCT
   A_SCLight : BOOL ;	//Screen light
   A_SCDark : BOOL ;	//Screen darkening
   A_KeyDisable : BOOL ;	//Key disable
   A_ClearCanAl : BOOL ;	//Clear cancel alarms
   A_ClearRecAl : BOOL ;	//Clear recall alarms
   f0_5 : BOOL ;
   f0_6 : BOOL ;
   A_ActWCS : BOOL ;	//Actual value in WCS 0=MCS
   A_PLCExtViewerReject : BOOL ;	//External viewer reject
   A_PLCExtViewerMode : BOOL ;	//External viewer mode
   f1_2 : BOOL ;
   f1_3 : BOOL ;
   f1_4 : BOOL ;
   f1_5 : BOOL ;
   f1_6 : BOOL ;
   f1_7 : BOOL ;
   A_1stError1 : WORD ;	//1st error HIGRAPH
   A_1stError2 : WORD ;	//1st error HIGRAPH
   A_ASpi1percent : BYTE ;	//Analog spindle 1:
   A_ASpi2percent : BYTE ;
   A_MCPChan : BYTE ;
   A_OEM1 : BOOL ;
   A_OEM2 : BOOL ;
   A_AToolMeas : BOOL ;	//AutoToolMeasure
   f9_3 : BOOL ;
   f9_4 : BOOL ;
   f9_5 : BOOL ;
   f9_6 : BOOL ;
   f9_7 : BOOL ;
   A_Hardkey : BYTE ;	//PLC Hardkeys
   f11 : BYTE ;	//Reserved for hardkeys
   f12_0 : BOOL ;
   f12_1 : BOOL ;
   A_COM2 : BOOL ;
   A_COM1 : BOOL ;
   A_V24stop : BOOL ;
   A_V24ext : BOOL ;
   A_V24off : BOOL ;
   A_V24on : BOOL ;
   A_TeachDisable : BOOL ;
   f13_1 : BOOL ;
   f13_2 : BOOL ;
   f13_3 : BOOL ;
   f13_4 : BOOL ;
   A_PPdeload : BOOL ;
   A_PPload : BOOL ;
   A_PPsel : BOOL ;
   A_V24Index1 : BYTE ;
   A_V24Index2 : BYTE ;
   A_V24NoFile1 : BYTE ;
   A_V24NoFile2 : BYTE ;
   A_res18 : BYTE ;
   A_res19 : BYTE ;	//Message counter
   f20_0 : BOOL ;
   E_SCDark : BOOL ;	//Screen darkening
   E_Cancel : BOOL ;	//Cancel
   E_CanCleared : BOOL ;	//Cancel alarms cleared
   E_RecCleared : BOOL ;	//Recall alarms cleared
   f20_5 : BOOL ;	//res. Language
   E_SimActiv : BOOL ;	//Simulation active
   E_ActWCS : BOOL ;	//Switchover MCS/WCS 0=MCS
   E_ActivWA : BYTE ;
   E_Chan : BYTE ;	//Channel displayed
   f23 : BYTE ;
   E_V24Err : BOOL ;
   E_V24OK : BOOL ;
   E_V24COM2 : BOOL ;
   E_V24COM1 : BOOL ;
   E_V24stop : BOOL ;
   E_V24ext : BOOL ;
   E_V24off : BOOL ;
   E_V24on : BOOL ;
   E_V24Error : BYTE ;	//V24: Error Byte
   E_res26_0 : BOOL ;	//Reserved
   E_PPOK : BOOL ;	//Part program status OK
   E_PPErr : BOOL ;	//Part program status Error
   E_PPAct : BOOL ;	//Part program status active
   f26_4 : BOOL ;	//Reserved
   E_PPdeload : BOOL ;	//Part program status deloading
   E_PPload : BOOL ;	//Part program status loading
   E_PPsel : BOOL ;	//Part program status selecting
   E_PPError : BYTE ;	//Part program status Error
   A_PictNo : INT ;
   A_PictOn : BOOL ;
   A_PictOff : BOOL ;
   f30_2 : BOOL ;
   f30_3 : BOOL ;
   f30_4 : BOOL ;
   f30_5 : BOOL ;
   f30_6 : BOOL ;
   f30_7 : BOOL ;
   E_PictOK : BOOL ;
   E_PictOn : BOOL ;
   E_PictAct : BOOL ;
   E_PictOff : BOOL ;
   E_PictErr : BOOL ;
   f31_5 : BOOL ;
   f31_6 : BOOL ;
   E_NotAct : BOOL ;
   A_FuncNo : BYTE ;
   A_Par1 : BYTE ;
   A_Par2 : BYTE ;
   A_Par3 : BYTE ;
   E_FuncErr : BYTE ;
   f37 : BYTE ;
   f38 : BYTE ;
   f39 : BYTE ;
   res40 : ARRAY  [0 .. 9 ] OF BYTE ;
   MMC2 : STRUCT
    A_SCLight : BOOL ;	//Screen light
    A_SCDark : BOOL ;	//Screen darkening
    A_KeyDisable : BOOL ;	//Key disable
    A_ClearCanAl : BOOL ;	//Clear cancel alarms
    A_ClearRecAl : BOOL ;	//Clear recall alarms
    f0_5 : BOOL ;
    f0_6 : BOOL ;
    A_ActWCS : BOOL ;	//Actual value in WCS 0=MCS
    A_1stError1 : WORD ;	//1st error HIGRAPH
    A_1stError2 : WORD ;	//1st error HIGRAPH
    A_ASpi1percent : BYTE ;	//Analog spindle 1:
    A_ASpi2percent : BYTE ;
    A_MCPChan : BYTE ;
    A_OEM1 : BOOL ;
    A_OEM2 : BOOL ;
    A_AToolMeas : BOOL ;	//AutoToolMeasure
    f9_3 : BOOL ;
    f9_4 : BOOL ;
    f9_5 : BOOL ;
    f9_6 : BOOL ;
    f9_7 : BOOL ;
    A_Hardkey : BYTE ;	//PLC Hardkeys
    f11 : BYTE ;	//Reserved for hardkeys
    f12_0 : BOOL ;
    f12_1 : BOOL ;
    A_COM2 : BOOL ;
    A_COM1 : BOOL ;
    A_V24stop : BOOL ;
    A_V24ext : BOOL ;
    A_V24off : BOOL ;
    A_V24on : BOOL ;
    f13_0 : BOOL ;
    f13_1 : BOOL ;
    f13_2 : BOOL ;
    f13_3 : BOOL ;
    f13_4 : BOOL ;
    A_PPdeload : BOOL ;
    A_PPload : BOOL ;
    A_PPsel : BOOL ;
    A_V24Index1 : BYTE ;
    A_V24Index2 : BYTE ;
    A_V24NoFile1 : BYTE ;
    A_V24NoFile2 : BYTE ;
    A_res18 : BYTE ;
    A_res19 : BYTE ;	//Message counter
    f20_0 : BOOL ;
    E_SCDark : BOOL ;	//Screen darkening
    E_Cancel : BOOL ;	//Cancel
    E_CanCleared : BOOL ;	//Cancel alarms cleared
    E_RecCleared : BOOL ;	//Recall alarms cleared
    f20_5 : BOOL ;	//res. Language
    E_SimActiv : BOOL ;	//Simulation active
    E_ActWCS : BOOL ;	//Switchover MCS/WCS 0=MCS
    E_ActivWA : BYTE ;
    E_Chan : BYTE ;	//Channel displayed
    f23 : BYTE ;
    E_V24Err : BOOL ;
    E_V24OK : BOOL ;
    E_V24COM2 : BOOL ;
    E_V24COM1 : BOOL ;
    E_V24stop : BOOL ;
    E_V24ext : BOOL ;
    E_V24off : BOOL ;
    E_V24on : BOOL ;
    E_V24Error : BYTE ;	//V24: Error Byte
    E_res26_0 : BOOL ;	//Reserved
    E_PPOK : BOOL ;	//Part program status OK
    E_PPErr : BOOL ;	//Part program status Error
    E_PPAct : BOOL ;	//Part program status active
    f26_4 : BOOL ;	//Reserved
    E_PPdeload : BOOL ;	//Part program status deloading
    E_PPload : BOOL ;	//Part program status loading
    E_PPsel : BOOL ;	//Part program status selecting
    E_PPError : BYTE ;	//Part program status Error
    A_PictNo : INT ;
    A_PictOn : BOOL ;
    A_PictOff : BOOL ;
    f30_2 : BOOL ;
    f30_3 : BOOL ;
    f30_4 : BOOL ;
    f30_5 : BOOL ;
    f30_6 : BOOL ;
    f30_7 : BOOL ;
    E_PictOK : BOOL ;
    E_PictOn : BOOL ;
    E_PictAct : BOOL ;
    E_PictOff : BOOL ;
    E_PictErr : BOOL ;
    f31_5 : BOOL ;
    f31_6 : BOOL ;
    E_NotAct : BOOL ;
    A_FuncNo : BYTE ;
    A_Par1 : BYTE ;
    A_Par2 : BYTE ;
    A_Par3 : BYTE ;
    E_FuncErr : BYTE ;
    f37 : BYTE ;
    f38 : BYTE ;
    f39 : BYTE ;
    res40 : ARRAY  [0 .. 9 ] OF BYTE ;
   END_STRUCT ;	//M to N
   ONL_REQUEST : WORD ;
   ONL_CONFIRM : WORD ;
   PAR_CLIENT_IDENT : WORD ;
   PAR_MMC_TYP : BYTE ;
   PAR_MSTT_ADR : BYTE ;
   PAR_STATUS : BYTE ;
   PAR_Z_INFO : BYTE ;
   MtoNAlive : WORD ;
   f112 : BYTE ;
   ParOpKeyAdr : BYTE ;
   ParTcuIndex : BYTE ;
   f115 : BYTE ;
   Tcu1KeyAdr : BYTE ;
   Tcu2KeyAdr : BYTE ;
   Tcu1Index : BYTE ;
   Tcu2Index : BYTE ;
   MMC1_CLIENT_IDENT : WORD ;
   MMC1_TYP : BYTE ;
   MMC1_MSTT_ADR : BYTE ;
   MMC1_STATUS : BYTE ;
   MMC1_Z_INFO : BYTE ;
   MMC1_SHIFT_LOCK : BOOL ;
   MMC1_MSTT_SHIFT_LOCK : BOOL ;
   MMC1_ACTIVE_REQ : BOOL ;
   MMC1_ACTIVE_PERM : BOOL ;
   MMC1_ACTIVE_CHANGED : BOOL ;
   MMC1_CHANGED_DENIED : BOOL ;
   MMC1_TCU_SHIFT_LOCK : BOOL ;
   f127 : BYTE ;
   MMC1_TRANS_DB : WORD ;
   MMC2_CLIENT_IDENT : WORD ;
   MMC2_TYP : BYTE ;
   MMC2_MSTT_ADR : BYTE ;
   MMC2_STATUS : BYTE ;
   MMC2_Z_INFO : BYTE ;
   MMC2_SHIFT_LOCK : BOOL ;
   MMC2_MSTT_SHIFT_LOCK : BOOL ;
   MMC2_ACTIVE_REQ : BOOL ;
   MMC2_ACTIVE_PERM : BOOL ;
   MMC2_ACTIVE_CHANGED : BOOL ;
   MMC2_CHANGED_DENIED : BOOL ;
   MMC2_TCU_SHIFT_LOCK : BOOL ;
   f137 : BYTE ;
   MMC2_TRANS_DB : WORD ;
   A_Subtype : INT ;	//for Codecarrier Input from PLC
   A_Duplo : INT ;
   A_Ident : STRING  [32 ];
   A_Tnumber : INT ;
   A_MagazinePlace : INT ;
   A_MagazinePlaceType : INT ;
   A_ToolSize_Upper : BYTE ;
   A_ToolSize_Down : BYTE ;
   A_ToolSize_Left : BYTE ;
   A_ToolSize_Right : BYTE ;
   A_Channel : BYTE ;
   A_LoadingPlace : BYTE ;
   A_Magazine : INT ;
   A_Unit : BYTE ;
   A_NCU_Index : BYTE ;
   A_FileIndex : INT ;
   A_ActiveEnable : BOOL ;
   A_Override : BOOL ;
   A_LoadTool : BOOL ;
   A_DeleteTool : BOOL ;
   E_Subtype : INT ;	//for Codecarrier Output to PLC
   E_Duplo : INT ;
   E_Ident : STRING  [32 ];
   E_Tnumber : INT ;
   E_ToolState : INT ;
   E_MagazinePlaceType : INT ;
   E_ToolSize_Upper : BYTE ;
   E_ToolSize_Down : BYTE ;
   E_ToolSize_Left : BYTE ;
   E_ToolSize_Right : BYTE ;
   E_Magazine : INT ;
   E_MagazinePlace : INT ;
   A_ReqMMC1 : BOOL ;	//for Codecarrier Request MMC-Interface1
   A_ReqMMC2 : BOOL ;	//for Codecarrier Request MMC-Interface2
   A_K_Code : BYTE ;
   E_Done : BOOL ;
   E_Error : BOOL ;
   E_Active : BOOL ;	// CodeCarrierReadEnable : BOOL;
// CodeCarrierWriteEnable : BOOL;
   E_K_CodeError : BYTE ;	//Identify for Error_Code
   E_Error_Code : INT ;
   E_Req : BOOL ;	//for Positioning
   f257 : BYTE ;
   A_Done : BOOL ;
   A_Error : BOOL ;
   A_Active : BOOL ;
   f258_3 : BOOL ;
   f258_4 : BOOL ;
   f258_5 : BOOL ;
   f258_6 : BOOL ;
   f258_7 : BOOL ;
   E_TDC_Read : BOOL ;
   E_TDC_Write : BOOL ;
   E_TDC_Cancel : BOOL ;
   A_Error_Code : INT ;
   E_PMagazine : INT ;
   E_PMagazinePlace : INT ;
   E_PTnumber : INT ;	//TPM-Data
   A_TPMStatus : INT ;
   A_TPMCounter : ARRAY  [1 .. 32 ] OF DINT ;
   A_HWeelSimOvr : BYTE ;
   f399 : BYTE ;
   A_SimOvr : INT ;
  END_STRUCT ;	
BEGIN
END_DATA_BLOCK

DATA_BLOCK "MSTT_1"	// DB 81
AUTHOR : SEDIN
VERSION : 0.1
  STRUCT
   B_AUTO : BOOL ;	//Клавиша "AUTO"
   B_MDA : BOOL ;	//Клавиша "MDA"
   B_TEACHIN : BOOL ;	//Клавиша "TEACH IN"
   B_JOG : BOOL ;	//Клавиша "JOG"
   S_Feed2Over0 : BOOL ;	//Корректор скорости подачи, бит 0
   S_Feed2Over1 : BOOL ;	//Корректор скорости подачи, бит 1
   S_Feed2Over2 : BOOL ;	//Корректор скорости подачи, бит 2
   S_Feed2Over3 : BOOL ;	//Корректор скорости подачи, бит 3
   B_INC1 : BOOL ;	//Клавиша "1 INC"
   B_INC10 : BOOL ;	//Клавиша "10 INC"
   B_INC100 : BOOL ;	//Клавиша "100 INC"
   B_INC1000 : BOOL ;	//Клавиша "1000 INC"
   B_INC10000 : BOOL ;	//Клавиша "10000 INC"
   B_INCVar : BOOL ;	//Клавиша "Var. INC"
   B_REF : BOOL ;	//Клавиша "REF"
   B_REPOS : BOOL ;	//Клавиша "REPOS"
   B_NCStop : BOOL ;	//Клавиша "*NC Stop"
   B_NCStart : BOOL ;	//Клавиша "NC Start"
   B_Chan1Stop : BOOL ;	//Клавиша "*Стоп в канале 1"
   B_Chan1Start : BOOL ;	//Клавиша "Старт в канале 1"
   B_Chan2Stop : BOOL ;	//Клавиша "*Стоп в канале 2"
   B_Chan2Start : BOOL ;	//Клавиша "Старт в канале 2"
   S_Pos2 : BOOL ;	//Переключатель, позиция 2
   S_Pos0 : BOOL ;	//Переключатель, позиция 0
   S_Feed1Over0 : BOOL ;	//Корректор скорости подачи, бит 0
   S_Feed1Over1 : BOOL ;	//Корректор скорости подачи, бит 1
   S_Feed1Over2 : BOOL ;	//Корректор скорости подачи, бит 2
   S_Feed1Over3 : BOOL ;	//Корректор скорости подачи, бит 3
   S_Feed1Over4 : BOOL ;	//Корректор скорости подачи, бит 4
   B_SingleBlock : BOOL ;	//Клавиша "Single Block"
   S_Pos1 : BOOL ;	//Переключатель, позиция 1
   B_Reset : BOOL ;	//Клавиша "Reset"
   B_R10 : BOOL ;	//Клавиша ""
   B_Lub1 : BOOL ;	//Клавиша "Прокачка ИСС 1"
   B_Xminus : BOOL ;	//Клавиша "X-"
   B_R1 : BOOL ;	//Клавиша ""
   S_Pos3 : BOOL ;	//Переключатель, позиция 3
   B_R14 : BOOL ;	//Клавиша ""
   B_R13 : BOOL ;	//Клавиша ""
   B_R15 : BOOL ;	//Клавиша ""
   B_Xplus : BOOL ;	//Клавиша "X+"
   B_Zminus : BOOL ;	//Клавиша "Z-"
   B_R9 : BOOL ;	//Клавиша ""
   B_Light1 : BOOL ;	//Клавиша "Включение освещения на станке 1"
   B_R12 : BOOL ;	//Клавиша ""
   B_Rapid1 : BOOL ;	//Клавиша "Ускоренный ход 1"
   B_R3 : BOOL ;	//Клавиша ""
   B_Zplus : BOOL ;	//Клавиша "Z+"
   not_used : BOOL ;
   B_T15 : BOOL ;	//Клавиша ""
   B_T14 : BOOL ;	//Клавиша ""
   B_T13 : BOOL ;	//Клавиша ""
   B_T12 : BOOL ;	//Клавиша ""
   B_Light2 : BOOL ;	//Клавиша "Включение освещения на станке 2"
   B_T10 : BOOL ;	//Клавиша ""
   B_T9 : BOOL ;	//Клавиша ""
   B_Wminus : BOOL ;	//Клавиша "W-"
   B_Lub2 : BOOL ;	//Клавиша "Прокачка ИСС 2"
   B_Uminus : BOOL ;	//Клавиша "U-"
   B_Rapid2 : BOOL ;	//Клавиша "Ускоренный ход 2"
   B_UPlus : BOOL ;	//Клавиша "U+"
   B_T3 : BOOL ;	//Клавиша ""
   B_Wplus : BOOL ;	//Клавиша "W+"
   B_T1 : BOOL ;	//Клавиша ""
   not_used1 : BYTE ;
   not_used2 : BYTE ;
   KT1 : BOOL ;
   KT2 : BOOL ;
   KT3 : BOOL ;
   KT4 : BOOL ;
   KT5 : BOOL ;
   KT6 : BOOL ;
   KT7 : BOOL ;
   KT8 : BOOL ;
   KT9 : BOOL ;
   not_used3 : BOOL ;
   not_used4 : BOOL ;
   not_used5 : BOOL ;
   not_used6 : BOOL ;
   not_used7 : BOOL ;
   not_used8 : BOOL ;
   not_used9 : BOOL ;
   not_used10 : BYTE ;
   X31_pin_10 : BOOL ;
   X31_pin_9 : BOOL ;
   X31_pin_8 : BOOL ;
   X31_pin_7 : BOOL ;
   X31_pin_6 : BOOL ;
   not_used11 : BOOL ;
   not_used12 : BOOL ;
   not_used13 : BOOL ;
   Handwheel_1 : WORD ;
   Handwheel_2 : WORD ;
   L_AUTO : BOOL ;	//Светодиод "AUTO"
   L_MDA : BOOL ;	//Светодиод "MDA"
   L_TEACHIN : BOOL ;	//Светодиод "TEACH IN"
   L_JOG : BOOL ;	//Светодиод "JOG"
   L_INC1 : BOOL ;	//Светодиод "1 INC"
   L_INC10 : BOOL ;	//Светодиод "10 INC"
   L_INC100 : BOOL ;	//Светодиод "100 INC"
   L_INC1000 : BOOL ;	//Светодиод "1000 INC"
   L_INC10000 : BOOL ;	//Светодиод "10000 INC"
   L_INCVar : BOOL ;	//Светодиод "Var. INC"
   L_REF : BOOL ;	//Светодиод "REF"
   L_REPOS : BOOL ;	//Светодиод "REPOS"
   L_NCStop : BOOL ;	//Светодиод "*NC Stop"
   L_NCStart : BOOL ;	//Светодиод "NC Start"
   L_Chan1Stop : BOOL ;	//Светодиод "*Стоп в канале 1"
   L_Chan1Start : BOOL ;	//Светодиод "Старт в канале 1"
   L_Chan2Stop : BOOL ;	//Светодиод "*Стоп в канале 2"
   L_Chan2Start : BOOL ;	//Светодиод "Старт в канале 2"
   L_SingleBlock : BOOL ;	//Светодиод "Single Block"
   L_R10 : BOOL ;	//Светодиод ""
   L_Lub1 : BOOL ;	//Светодиод "Прокачка ИСС 1"
   L_Xminus : BOOL ;	//Светодиод "X-"
   L_R1 : BOOL ;	//Светодиод ""
   L_R13 : BOOL ;	//Светодиод ""
   L_R15 : BOOL ;	//Светодиод ""
   L_Xplus : BOOL ;	//Светодиод "X+"
   L_Zminus : BOOL ;	//Светодиод "Z-"
   L_R9 : BOOL ;	//Светодиод ""
   L_Light1 : BOOL ;	//Светодиод "Включение освещения на станке 1"
   L_R12 : BOOL ;	//Светодиод ""
   L_Rapid1 : BOOL ;	//Светодиод "Ускоренный ход 1"
   L_R3 : BOOL ;	//Светодиод ""
   L_Zplus : BOOL ;	//Светодиод "Z+"
   L_T15 : BOOL ;	//Светодиод ""
   L_T14 : BOOL ;	//Светодиод ""
   L_T13 : BOOL ;	//Светодиод ""
   L_T12 : BOOL ;	//Светодиод ""
   L_Light2 : BOOL ;	//Светодиод "Включение освещения на станке 2"
   L_T10 : BOOL ;	//Светодиод ""
   L_T9 : BOOL ;	//Светодиод ""
   L_Wminus : BOOL ;	//Светодиод "W-"
   L_Lub2 : BOOL ;	//Светодиод "Прокачка ИСС 2"
   L_Uminus : BOOL ;	//Светодиод "U-"
   L_Rapid2 : BOOL ;	//Светодиод "Ускоренный ход 2"
   L_UPlus : BOOL ;	//Светодиод "U+"
   L_T3 : BOOL ;	//Светодиод ""
   L_Wplus : BOOL ;	//Светодиод "W+"
   L_T1 : BOOL ;	//Светодиод ""
   L_R14 : BOOL ;	//Unused
   L_Reset : BOOL ;	//Светодиод "Reset"
   L_not_used1 : BOOL ;	//Not used
   L_not_used2 : BOOL ;	//Not used
   L_not_used3 : BOOL ;	//Not used
   L_not_used4 : BOOL ;	//Not used
   L_not_used5 : BOOL ;	//Not used
   L_not_used6 : BOOL ;	//Not used
   KT_OUT_1 : BOOL ;	//Not used
   KT_OUT_2 : BOOL ;	//Not used
   KT_OUT_3 : BOOL ;	//Not used
   KT_OUT_4 : BOOL ;	//Not used
   KT_OUT_5 : BOOL ;	//Not used
   KT_OUT_6 : BOOL ;	//Not used
   L_not_used14 : BOOL ;	//Not used
   L_not_used15 : BOOL ;	//Not used
   StatSend : DWORD ;	//Состояние передачи на станочный пульт
   StatRec : DWORD ;	//Состояние приема на станочный пульт
  END_STRUCT ;	
BEGIN
END_DATA_BLOCK

DATA_BLOCK "MSTT_2"	// DB 82
AUTHOR : SEDIN
VERSION : 0.1
  STRUCT
   B_AUTO : BOOL ;	//Клавиша "AUTO"
   B_MDA : BOOL ;	//Клавиша "MDA"
   B_Unclump : BOOL ;	//Клавиша "Отжим детали"
   B_Clamp : BOOL ;	//Клавиша "Прижим детали"
   S_Feed3Over0 : BOOL ;	//Корректор скорости подачи, бит 0
   S_Feed3Over1 : BOOL ;	//Корректор скорости подачи, бит 1
   S_Feed3Over2 : BOOL ;	//Корректор скорости подачи, бит 2
   S_Feed3Over3 : BOOL ;	//Корректор скорости подачи, бит 3
   B_INC1 : BOOL ;	//Клавиша "1 INC"
   B_INC10 : BOOL ;	//Клавиша "10 INC"
   B_INC100 : BOOL ;	//Клавиша "100 INC"
   B_SpindleJog : BOOL ;	//Клавиша "Толчковый режим главного привода"
   B_INC10000 : BOOL ;	//Клавиша "10000 INC"
   B_Unchuck : BOOL ;	//Клавиша "Разжим детали"
   B_REF : BOOL ;	//Клавиша "REF"
   B_Chuck : BOOL ;	//Клавиша "Зажим детали"
   B_SpindleStop : BOOL ;	//Клавиша "Стоп планшайбы"
   B_SpindleCW : BOOL ;	//Клавиша "Пуск планшайбы по часовой"
   B_Chan3Stop : BOOL ;	//Клавиша "*Стоп в канале 3"
   B_Chan3Start : BOOL ;	//Клавиша "Старт в канале 3"
   B_Chan4Stop : BOOL ;	//Клавиша "*Стоп в канале 4"
   B_Chan4Start : BOOL ;	//Клавиша "Старт в канале 4"
   S_Pos2 : BOOL ;	//Переключатель, позиция 2
   S_Pos0 : BOOL ;	//Переключатель, позиция 0
   S_Feed4Over0 : BOOL ;	//Корректор скорости подачи, бит 0
   S_Feed4Over1 : BOOL ;	//Корректор скорости подачи, бит 1
   S_Feed4Over2 : BOOL ;	//Корректор скорости подачи, бит 2
   S_Feed4Over3 : BOOL ;	//Корректор скорости подачи, бит 3
   S_Feed4Over4 : BOOL ;	//Корректор скорости подачи, бит 4
   B_SpindleCCW : BOOL ;	//Клавиша "Пуск планшайбы против часовой"
   S_Pos1 : BOOL ;	//Переключатель, позиция 1
   B_Reset : BOOL ;	//Клавиша "Reset"
   B_R10 : BOOL ;	//Клавиша ""
   B_Lub3 : BOOL ;	//Клавиша "Прокачка ИСС 3"
   B_X1minus : BOOL ;	//Клавиша "X1-"
   B_R1 : BOOL ;	//Клавиша ""
   S_Pos3 : BOOL ;	//Переключатель, позиция 3
   B_R14 : BOOL ;	//Клавиша ""
   B_R13 : BOOL ;	//Клавиша ""
   B_HHU : BOOL ;	//Клавиша "Активизация выносного пульта"
   B_X1plus : BOOL ;	//Клавиша "X1+"
   B_Z1minus : BOOL ;	//Клавиша "Z1-"
   B_R9 : BOOL ;	//Клавиша ""
   B_R11 : BOOL ;	//Клавиша ""
   B_R12 : BOOL ;	//Клавиша ""
   B_Rapid3 : BOOL ;	//Клавиша "Ускоренный ход 3"
   B_R3 : BOOL ;	//Клавиша ""
   B_Z1plus : BOOL ;	//Клавиша "Z1+"
   not_used : BOOL ;
   B_T15 : BOOL ;	//Клавиша ""
   B_T14 : BOOL ;	//Клавиша ""
   B_T13 : BOOL ;	//Клавиша ""
   B_T12 : BOOL ;	//Клавиша ""
   B_T11 : BOOL ;	//Клавиша ""
   B_T10 : BOOL ;	//Клавиша ""
   B_T9 : BOOL ;	//Клавиша ""
   B_W1minus : BOOL ;	//Клавиша "W1-"
   B_Lub4 : BOOL ;	//Клавиша "Прокачка ИСС 4"
   B_U1minus : BOOL ;	//Клавиша "U1-"
   B_Rapid4 : BOOL ;	//Клавиша "Ускоренный ход 4"
   B_U1Plus : BOOL ;	//Клавиша "U1+"
   B_T3 : BOOL ;	//Клавиша ""
   B_W1plus : BOOL ;	//Клавиша "W1+"
   B_T1 : BOOL ;	//Клавиша ""
   not_used1 : BYTE ;
   not_used11 : BYTE ;
   KT1 : BOOL ;
   KT2 : BOOL ;
   KT3 : BOOL ;
   KT4 : BOOL ;
   KT5 : BOOL ;
   KT6 : BOOL ;
   KT7 : BOOL ;
   KT8 : BOOL ;
   KT9 : BOOL ;
   not_used3 : BOOL ;
   not_used4 : BOOL ;
   not_used5 : BOOL ;
   not_used6 : BOOL ;
   not_used7 : BOOL ;
   not_used8 : BOOL ;
   not_used9 : BOOL ;
   not_used10 : BYTE ;
   X31_pin_10 : BOOL ;
   X31_pin_9 : BOOL ;
   X31_pin_8 : BOOL ;
   X31_pin_7 : BOOL ;
   X31_pin_6 : BOOL ;
   not_used111 : BOOL ;
   not_used12 : BOOL ;
   not_used13 : BOOL ;
   Handwheel_1 : WORD ;
   Handwheel_2 : WORD ;
   L_AUTO : BOOL ;	//Светодиод "AUTO"
   L_MDA : BOOL ;	//Светодиод "MDA"
   L_Unclump : BOOL ;	//Светодиод "Отжим детали"
   L_Clamp : BOOL ;	//Светодиод "Прижим детали"
   L_INC1 : BOOL ;	//Светодиод "1 INC"
   L_INC10 : BOOL ;	//Светодиод "10 INC"
   L_INC100 : BOOL ;	//Светодиод "100 INC"
   L_SpindleJog : BOOL ;	//Светодиод "Толчковый режим главного привода"
   L_INC10000 : BOOL ;	//Светодиод "10000 INC"
   L_Unchuck : BOOL ;	//Светодиод "Разжим детали"
   L_REF : BOOL ;	//Светодиод "REF"
   L_Chuck : BOOL ;	//Светодиод "Зажим детали"
   L_SpindleStop : BOOL ;	//Светодиод "Стоп  планшайбы"
   L_SpindleCW : BOOL ;	//Светодиод "Пуск планшайбы по часовой"
   L_Chan3Stop : BOOL ;	//Светодиод "*Стоп в канале 3"
   L_Chan3Start : BOOL ;	//Светодиод "Старт в канале 3"
   L_Chan4Stop : BOOL ;	//Светодиод "*Стоп в канале 4"
   L_Chan4Start : BOOL ;	//Светодиод "Старт в канале 4"
   L_SpindleCCW : BOOL ;	//Светодиод "Пуск планшайбы против часовой"
   L_R10 : BOOL ;	//Светодиод ""
   L_Lub3 : BOOL ;	//Светодиод "Прокачка ИСС 3"
   L_X1minus : BOOL ;	//Светодиод "X1-"
   L_R1 : BOOL ;	//Светодиод ""
   L_R13 : BOOL ;	//Светодиод ""
   L_HHU : BOOL ;	//Светодиод "Активизация выносного пульта"
   L_X1plus : BOOL ;	//Светодиод "X1+"
   L_Z1minus : BOOL ;	//Светодиод "Z1-"
   L_R9 : BOOL ;	//Светодиод ""
   L_R11 : BOOL ;	//Светодиод ""
   L_R12 : BOOL ;	//Светодиод ""
   L_Rapid3 : BOOL ;	//Светодиод "Ускоренный ход 3"
   L_R3 : BOOL ;	//Светодиод ""
   L_Z1plus : BOOL ;	//Светодиод "Z1+"
   L_T15 : BOOL ;	//Светодиод ""
   L_T14 : BOOL ;	//Светодиод ""
   L_T13 : BOOL ;	//Светодиод ""
   L_T12 : BOOL ;	//Светодиод ""
   L_T11 : BOOL ;	//Светодиод ""
   L_T10 : BOOL ;	//Светодиод ""
   L_T9 : BOOL ;	//Светодиод ""
   L_W1minus : BOOL ;	//Светодиод "W1-"
   L_Lub4 : BOOL ;	//Светодиод "Прокачка ИСС 4"
   L_U1minus : BOOL ;	//Светодиод "U1-"
   L_Rapid4 : BOOL ;	//Светодиод "Ускоренный ход 4"
   L_U1Plus : BOOL ;	//Светодиод "U1+"
   L_T3 : BOOL ;	//Светодиод ""
   L_W1plus : BOOL ;	//Светодиод "W1+"
   L_T1 : BOOL ;	//Светодиод ""
   L_R14 : BOOL ;	//Unused
   L_Reset : BOOL ;	//Светодиод "Reset"
   L_not_used1 : BOOL ;	//Not used
   L_not_used2 : BOOL ;	//Not used
   L_not_used3 : BOOL ;	//Not used
   L_not_used4 : BOOL ;	//Not used
   L_not_used5 : BOOL ;	//Not used
   L_not_used6 : BOOL ;	//Not used
   KT_OUT_1 : BOOL ;	//Not used
   KT_OUT_2 : BOOL ;	//Not used
   KT_OUT_3 : BOOL ;	//Not used
   KT_OUT_4 : BOOL ;	//Not used
   KT_OUT_5 : BOOL ;	//Not used
   KT_OUT_6 : BOOL ;	//Not used
   L_not_used14 : BOOL ;	//Not used
   L_not_used15 : BOOL ;	//Not used
   StatSend : DWORD ;	//Состояние передачи на станочный пульт
   StatRec : DWORD ;	//Состояние приема на станочный пульт
  END_STRUCT ;	
BEGIN
END_DATA_BLOCK

DATA_BLOCK "HHU"	// DB 83
AUTHOR : SEDIN
VERSION : 0.1
  STRUCT
   f0 : BYTE ;	//Резерв
   f1 : BYTE ;	//Резерв
   S5_U1 : BOOL ;	//Клавиша "U1"
   S1 : BOOL ;	//Клавиша ""
   S9_W1 : BOOL ;	//Клавиша "W1"
   S13_Inc_1 : BOOL ;	//Клавиша "Increment 1"
   S17_Handwheel : BOOL ;	//Клавиша "Handwheel"
   S6_U : BOOL ;	//Клавиша "U"
   S2_Minus : BOOL ;	//Клавиша "-"
   S10_W : BOOL ;	//Клавиша "W"
   S14_Inc_10 : BOOL ;	//Клавиша "Increment 10"
   S18_Inc_100 : BOOL ;	//Клавиша "Increment 100"
   S8_X1 : BOOL ;	//Клавиша "X1"
   S12_Z1 : BOOL ;	//Клавиша "Z1"
   S16_SpindleCW : BOOL ;	//Клавиша "Spindle Clock-wise"
   S20_SpindleJog : BOOL ;	//Клавиша "Spindle Jog"
   S7_X : BOOL ;	//Клавиша "X"
   S3_Plus : BOOL ;	//Клавиша "Plus"
   f4_0 : BOOL ;	//Not used
   f4_1 : BOOL ;	//Not used
   f4_2 : BOOL ;	//Not used
   f4_3 : BOOL ;	//Not used
   S4_Rapid : BOOL ;	//Клавиша "Rapid"
   S11_Z : BOOL ;	//Клавиша "Z"
   S15_SpindleCCW : BOOL ;	//Клавиша "Spindle Counterclock-wise"
   S19_SpindleStop : BOOL ;	//Клавиша "Spindle Stop"
   f5_0 : BOOL ;	//Not used
   S_FeedOver0 : BOOL ;	//Корректор скорости подачи, бит 0
   S_FeedOver1 : BOOL ;	//Корректор скорости подачи, бит 1
   S_FeedOver2 : BOOL ;	//Корректор скорости подачи, бит 2
   S_FeedOver3 : BOOL ;	//Корректор скорости подачи, бит 3
   S_FeedOver4 : BOOL ;	//Корректор скорости подачи, бит 4
   Keyswitch : BOOL ;	//Переключатель
   Acknowledgement : BOOL ;	//Квитирование цифровой индикации
   f6 : BYTE  := B#16#80;	//Резерв
   Selection_Line_1_2 : BOOL ;	//Selection line 1, 2 for HHU display
   Selection_Line_3_4 : BOOL ;	//Selection line 3, 4 for HHU display
   Reserved_7_2 : BOOL ;	//Not used
   Reserved_7_3 : BOOL ;	//Not used
   Reserved_7_4 : BOOL ;	//Not used
   Reserved_7_5 : BOOL ;	//Not used
   Reserved_7_6 : BOOL ;	//Not used
   New_Data : BOOL ;	//New data for selected line
   L5_U1 : BOOL ;	//Светодиод "U1"
   L11_Z : BOOL ;	//Светодиод "Z"
   L9_W1 : BOOL ;	//Светодиод "W1"
   L13_Inc_1 : BOOL ;	//Светодиод "Increment 1"
   L17_HandWheel : BOOL ;	//Светодиод "Handwheel"
   L6_U : BOOL ;	//Светодиод "U"
   L15_SpindleCCW : BOOL ;	//Светодиод "Spindle Counterclock-wise"
   L10_W : BOOL ;	//Светодиод "W"
   L14_Inc_10 : BOOL ;	//Светодиод "Increment 10"
   L18_Inc_100 : BOOL ;	//Светодиод "Increment 100"
   L8_X1 : BOOL ;	//Светодиод "X1"
   L12_Z1 : BOOL ;	//Светодиод "Z1"
   L16_SpindleCW : BOOL ;	//Светодиод "Spindle Clock-wise"
   L20_SpindleJog : BOOL ;	//Светодиод "Spindle Jog"
   L7_X : BOOL ;	//Светодиод "X"
   L19_SpindleStop : BOOL ;	//Светодиод "Spindle Stop"
   DataLine : ARRAY  [1 .. 16 ] OF //Индикация
   BYTE ;
   StatSend : DWORD ;	//Состояние передачи на пульт
   StatRec : DWORD ;	//Состояние приема на пульт
   Auxilary : ARRAY  [1 .. 8 ] OF //Вспомогательные
   BOOL ;
  END_STRUCT ;	
BEGIN
   S_FeedOver4 := TRUE;
END_DATA_BLOCK

DATA_BLOCK DB 105
AUTHOR : SEDIN
VERSION : 0.0
"Lathe_Modes"
BEGIN
END_DATA_BLOCK

DATA_BLOCK "Aux_Fun"	// DB 130
AUTHOR : SEDIN
VERSION : 0.1
  STRUCT
   MDyn : ARRAY  [0 .. 99 ] OF BOOL ;
   GAct : ARRAY  [1 .. 64 ] OF BYTE ;
  END_STRUCT ;	
BEGIN
END_DATA_BLOCK

DATA_BLOCK "NCVar_Pos"	// DB 140
VERSION : 0.0
  STRUCT
   N_measPos2 : STRUCT
    SYNTAX_ID : BYTE  := B#16#82;
    Area_Unit : BYTE  := B#16#1;
    Column : WORD  := W#16#6;
    Line : WORD ;
    BlockType : BYTE  := B#16#71;
    NumOfLine : BYTE  := B#16#1;
    DataType : BYTE  := B#16#F;
    Length : BYTE  := B#16#8;
   END_STRUCT ;
   C0_RP_rpa0 : STRUCT
    SYNTAX_ID : BYTE  := B#16#82;
    Area_Unit : BYTE  := B#16#40;
    Column : WORD  := W#16#1;
    Line : WORD ;
    BlockType : BYTE  := B#16#15;
    NumOfLine : BYTE  := B#16#1;
    DataType : BYTE  := B#16#F;
    Length : BYTE  := B#16#8;
   END_STRUCT ;
  END_STRUCT ;	
BEGIN
   N_measPos2.SYNTAX_ID := B#16#82;
   N_measPos2.Area_Unit := B#16#1;
   N_measPos2.Column := W#16#6;
   N_measPos2.BlockType := B#16#71;
   N_measPos2.NumOfLine := B#16#1;
   N_measPos2.DataType := B#16#F;
   N_measPos2.Length := B#16#8;
   C0_RP_rpa0.SYNTAX_ID := B#16#82;
   C0_RP_rpa0.Area_Unit := B#16#40;
   C0_RP_rpa0.Column := W#16#1;
   C0_RP_rpa0.BlockType := B#16#15;
   C0_RP_rpa0.NumOfLine := B#16#1;
   C0_RP_rpa0.DataType := B#16#F;
   C0_RP_rpa0.Length := B#16#8;
END_DATA_BLOCK

DATA_BLOCK "Share"	// DB 150
AUTHOR : SEDIN
VERSION : 0.1
  STRUCT
   Status : ARRAY  [0 .. 127 ] OF //Технологические данные
   BOOL  := FALSE;
   NumLathe : BYTE ;	//Порядковый номер станка
   StartCycle : BYTE ;	//Флаг начала цикла
   StopCycle : BYTE ;	//Флаг окончания цикла
   NumWheel : STRING  [10 ];	//Номер колеса
   NumMelt : STRING  [10 ];	//Номер плавки
   SideWheel : BYTE ;	//Код стороны колеса
   NumProgTrans : DWORD ;	//Номер программы обработки, переданной на станок
   NumProgFact : DWORD ;	//Номер фактической программы обработки
   CauseStop : BYTE ;	//Причина остановки программы
   YearStart : BYTE ;	//Год начала цикла
   MonthStart : BYTE ;	//Месяц начала цикла
   DayStart : BYTE ;	//День начала цикла
   HourStart : BYTE ;	//Час начала цикла
   MinStart : BYTE ;	//Минута начала цикла
   SecStart : BYTE ;	//Секунда начала цикла
   YearStop : BYTE ;	//Год окончания цикла
   MonthStop : BYTE ;	//Месяц окончания цикла
   DayStop : BYTE ;	//День начала цикла
   HourStop : BYTE ;	//Час окончания цикла
   MinStop : BYTE ;	//Минута окончания цикла
   SecStop : BYTE ;	//Секунда окончания цикла
   EstimTime : DWORD ;	//Расчетное время цикла
   FactTime : DWORD ;	//Фактическое время цикла
   ToolDate : ARRAY  [1 .. 6 ] OF //Данные инструмента
   STRUCT
    Number : BYTE ;	//Номер инструмента
    Channel : BYTE ;	//Номер канала
    Status : BYTE ;	//Статус
   END_STRUCT ;
  END_STRUCT ;	
BEGIN
END_DATA_BLOCK

DATA_BLOCK "CtrlE"	// DB 1000
TITLE = Datainterface Ctrl-Energy
AUTHOR : NUMERIK
FAMILY : _800D
NAME : CTRL_E
VERSION : 2.7
  STRUCT
   Profile : ARRAY  [1 .. 8 ] OF STRUCT
    ESaveOn : BOOL ;	// Activate energy-saving profile immediately
    ReloadT2 : BOOL ;	// Reload Prewarning time (T2)
    res0_2 : BOOL ;
    res0_3 : BOOL ;
    res0_4 : BOOL ;
    res0_5 : BOOL ;
    res0_6 : BOOL ;
    res0_7 : BOOL ;
    HmiESaveOn : BOOL ;	// HMI->PLC: Activate energy-saving profile immediately
    res1_1 : BOOL ;
    res1_2 : BOOL ;
    res1_3 : BOOL ;
    res1_4 : BOOL ;
    res1_5 : BOOL ;
    res1_6 : BOOL ;
    res1_7 : BOOL ;
    MasterCompSig : BOOL ;	// Master computer signal
    PlcUserSig : BOOL ;	// PLC user signal
    res2_2 : BOOL ;
    res2_3 : BOOL ;
    res2_4 : BOOL ;
    res2_5 : BOOL ;
    res2_6 : BOOL ;
    res2_7 : BOOL ;
    res3 : BYTE ;
    ESaveIsOn : BOOL ;	// Energy-saving state active
    T1Expired : BOOL ;	// Activation time T1 expired
    res4_2 : BOOL ;
    res4_3 : BOOL ;
    res4_4 : BOOL ;
    res4_5 : BOOL ;
    res4_6 : BOOL ;
    res4_7 : BOOL ;
    res5 : BYTE ;
    ActValT1 : INT ;	// T1 current value
    ActValT2 : INT ;	// T2 current value
    ESaveValid : BOOL ;	// HMI->PLC: Energy-saving profile valid
    ESaveOff : BOOL ;	// HMI->PLC: Deactivate energy-saving profileblock energy-saving profile
    res10_2 : BOOL ;
    res10_3 : BOOL ;
    res10_4 : BOOL ;
    res10_5 : BOOL ;
    res10_6 : BOOL ;
    res10_7 : BOOL ;
    CondOpPanel : BOOL ;	// HMI->PLC: Operator panel
    CondDataTransfer : BOOL ;	// HMI->PLC: Data transfer
    CondWindowChange : BOOL ;	// HMI->PLC: Window change
    res11_3 : BOOL ;
    res11_4 : BOOL ;
    res11_5 : BOOL ;
    res11_6 : BOOL ;
    res11_7 : BOOL ;
    CondMCP : BOOL ;	// HMI->PLC: Machine control panel
    res12_1 : BOOL ;
    res12_2 : BOOL ;
    res12_3 : BOOL ;
    res12_4 : BOOL ;
    res12_5 : BOOL ;
    res12_6 : BOOL ;
    res12_7 : BOOL ;
    CondNcChan1 : BOOL ;	// HMI->PLC: NC channel 1 in reset
    CondNcChan2 : BOOL ;	// HMI->PLC: NC channel 2 in reset
    CondNcChan3 : BOOL ;	// HMI->PLC: NC channel 3 in reset
    CondNcChan4 : BOOL ;	// HMI->PLC: NC channel 4 in reset
    CondNcChan5 : BOOL ;	// HMI->PLC: NC channel 5 in reset
    CondNcChan6 : BOOL ;	// HMI->PLC: NC channel 6 in reset
    CondNcChan7 : BOOL ;	// HMI->PLC: NC channel 7 in reset
    CondNcChan8 : BOOL ;	// HMI->PLC: NC channel 8 in reset
    CondNcChan9 : BOOL ;	// HMI->PLC: NC channel 9 in reset
    CondNcChan10 : BOOL ;	// HMI->PLC: NC channel 10 in reset
    res14_2 : BOOL ;
    res14_3 : BOOL ;
    res14_4 : BOOL ;
    res14_5 : BOOL ;
    res14_6 : BOOL ;
    res14_7 : BOOL ;
    CondMasterCompSig : BOOL ;	// HMI->PLC: Master computer signal
    CondPlcUserSig : BOOL ;	// HMI->PLC: PLC user signal
    res15_2 : BOOL ;
    res15_3 : BOOL ;
    res15_4 : BOOL ;
    res15_5 : BOOL ;
    res15_6 : BOOL ;
    res15_7 : BOOL ;
    PresetT1 : INT ;	// HMI->PLC: Activation time T1
    PresetT2 : INT ;	// HMI->PLC: Prewarning time T2
   END_STRUCT ;
  END_STRUCT ;	
BEGIN
   Profile[1].ESaveValid := TRUE;
   Profile[1].ESaveOff := TRUE;
   Profile[1].CondNcChan1 := TRUE;
   Profile[1].CondNcChan2 := TRUE;
   Profile[1].CondNcChan3 := TRUE;
   Profile[1].CondNcChan4 := TRUE;
   Profile[1].CondNcChan5 := TRUE;
   Profile[1].CondNcChan6 := TRUE;
   Profile[1].CondNcChan7 := TRUE;
   Profile[1].CondNcChan8 := TRUE;
   Profile[1].CondNcChan9 := TRUE;
   Profile[1].CondNcChan10 := TRUE;
   Profile[1].CondPlcUserSig := TRUE;
   Profile[1].PresetT1 := 60;
   Profile[1].PresetT2 := 120;
   Profile[2].ESaveValid := TRUE;
   Profile[2].ESaveOff := TRUE;
   Profile[2].CondMCP := TRUE;
   Profile[2].CondNcChan1 := TRUE;
   Profile[2].CondNcChan2 := TRUE;
   Profile[2].CondNcChan3 := TRUE;
   Profile[2].CondNcChan4 := TRUE;
   Profile[2].CondNcChan5 := TRUE;
   Profile[2].CondNcChan6 := TRUE;
   Profile[2].CondNcChan7 := TRUE;
   Profile[2].CondNcChan8 := TRUE;
   Profile[2].CondNcChan9 := TRUE;
   Profile[2].CondNcChan10 := TRUE;
   Profile[2].CondPlcUserSig := TRUE;
   Profile[2].PresetT1 := 120;
   Profile[2].PresetT2 := 300;
   Profile[3].ESaveValid := TRUE;
   Profile[3].ESaveOff := TRUE;
   Profile[3].CondOpPanel := TRUE;
   Profile[3].CondDataTransfer := TRUE;
   Profile[3].CondWindowChange := TRUE;
   Profile[3].CondMCP := TRUE;
   Profile[3].CondNcChan1 := TRUE;
   Profile[3].CondNcChan2 := TRUE;
   Profile[3].CondNcChan3 := TRUE;
   Profile[3].CondNcChan4 := TRUE;
   Profile[3].CondNcChan5 := TRUE;
   Profile[3].CondNcChan6 := TRUE;
   Profile[3].CondNcChan7 := TRUE;
   Profile[3].CondNcChan8 := TRUE;
   Profile[3].CondNcChan9 := TRUE;
   Profile[3].CondNcChan10 := TRUE;
   Profile[3].CondPlcUserSig := TRUE;
   Profile[3].PresetT1 := 600;
END_DATA_BLOCK

DATA_BLOCK "SentronPac"	// DB 1001
TITLE = Datainterface SentronPac
AUTHOR : NUMERIK
FAMILY : _800D
NAME : SENTRONP
VERSION : 2.7
  STRUCT
   ManualVal : BOOL ;	// Display of manual value
   SentronPacMach : BOOL ;	// Sentron PAC represented machine
   FeedInEnergyReadSP : BOOL ;	// Feed in energy read from Sentron PAC
   FeedBackEnergyReadSP : BOOL ;	// Feed back energy read from Sentron PAC
   res1 : BYTE ;
   MeasAct : BOOL ;	// Active measurement
   res3 : BYTE ;
   ManualValue : REAL ;	// Manual value
   ActivePowerItem : REAL ;	// Active power item
   ActiveEnergyItem : REAL ;	// Active energy item
   ReactiveEnergyItem : REAL ;	// Reactive energy item
  END_STRUCT ;	
BEGIN
END_DATA_BLOCK

ORGANIZATION_BLOCK "Cycle Execution"	// OB 1
TITLE = "Main Program Sweep (Cycle)"
VERSION : 0.1
VAR_TEMP
  OB1_EV_CLASS : BYTE ;	//Bits 0-3 = 1 (Coming event), Bits 4-7 = 1 (Event class 1)
  OB1_SCAN_1 : BYTE ;	//1 (Cold restart scan 1 of OB 1), 3 (Scan 2-n of OB 1)
  OB1_PRIORITY : BYTE ;	//Priority of OB Execution
  OB1_OB_NUMBR : BYTE ;	//1 (Organization block 1, OB1)
  OB1_RESERVED_1 : BYTE ;	//Reserved for system
  OB1_RESERVED_2 : BYTE ;	//Reserved for system
  OB1_PREV_CYCLE : INT ;	//Cycle time of previous OB1 scan (milliseconds)
  OB1_MIN_CYCLE : INT ;	//Minimum cycle time of OB1 (milliseconds)
  OB1_MAX_CYCLE : INT ;	//Maximum cycle time of OB1 (milliseconds)
  OB1_DATE_TIME : DATE_AND_TIME ;	//Date and time OB1 started
END_VAR
BEGIN
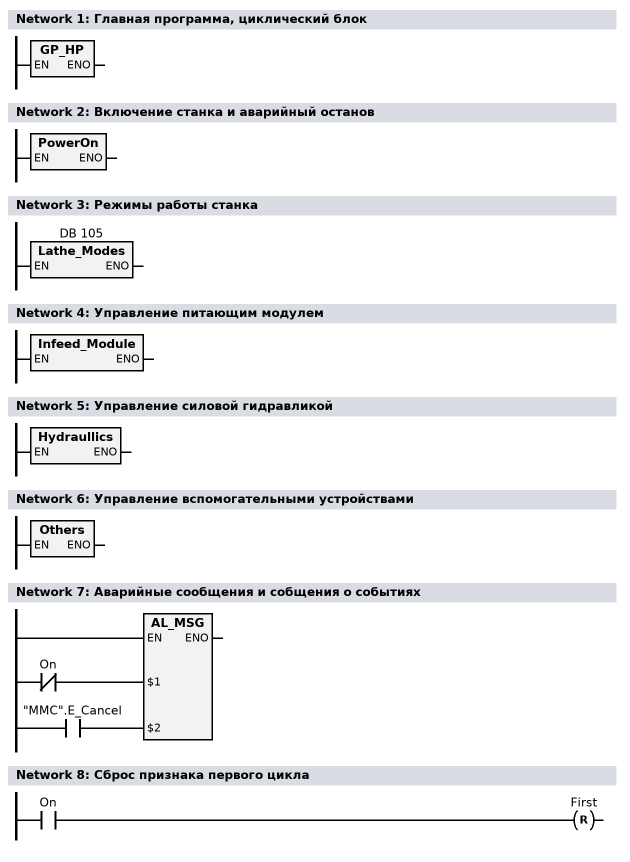
NETWORK
TITLE = Главная программа, циклический блок
      CALL  "GP_HP";
      NOP   0;
NETWORK
TITLE = Включение станка и аварийный останов
      CALL  "PowerOn";
      NOP   0;
NETWORK
TITLE = Режимы работы станка
      CALL  "Lathe_Modes" , DB 105;
      NOP   0;
NETWORK
TITLE = Управление питающим модулем
      CALL  "Infeed_Module";
      NOP   0;
NETWORK
TITLE = Управление силовой гидравликой
      CALL  "Hydraullics";
      NOP   0;
NETWORK
TITLE = Управление вспомогательными устройствами
      CALL  "Others";
      NOP   0;
NETWORK
TITLE = Аварийные сообщения и собщения о событиях
      AN    "On";
      =     L 20.0;
      BLD   103;
      A     "MMC".E_Cancel;
      =     L 20.1;
      BLD   103;
      CALL  "AL_MSG" (
           $1                       := L 20.0,
           $2                       := L 20.1);
      NOP   0;
NETWORK
TITLE = Сброс признака первого цикла
      A     "On";
      R     "First";
NETWORK
TITLE =
//      CALL  FC   150
      NOP   0;
END_ORGANIZATION_BLOCK

ORGANIZATION_BLOCK "HW_INT1"	// OB 40
VERSION : 1.0
VAR_TEMP
  OB40_EV_CLASS : BYTE ;
  OB40_STRT_INF : BYTE ;
  OB40_PRIORITY : BYTE ;
  OB40_OB_NUMBR : BYTE ;
  OB40_RESERVED_1 : BYTE ;
  OB40_MDL_ID : BYTE ;
  OB40_MDL_ADDR : INT ;
  OB40_POINT_ADDR : DWORD ;
  OB40_DATE_TIME : DATE_AND_TIME ;	//data for the Basic program
  GP_IRFromNCK : BOOL ;	//Interrupt from NCK
  GP_TM : BOOL ;	//Toolmanagment
  GP_InPosition : ARRAY  [1 .. 31 ] OF BOOL ;	//InPos Signal from FC15,16,18
  GP_AuxFunction : ARRAY  [1 .. 10 ] OF BOOL ;	//auxiliary functions
  GP_FMBlock : ARRAY  [1 .. 10 ] OF BOOL ;	//not used
//Insert User-data from here
END_VAR
BEGIN
NETWORK
TITLE =
      CALL  "GP_PRAL";
//Insert User program from here
END_ORGANIZATION_BLOCK

ORGANIZATION_BLOCK OB 82
TITLE = "I/O Point Fault"
VERSION : 1.0
VAR_TEMP
  OB82_EV_CLASS : BYTE ;	//16#39, Event class 3, Entering event state, Internal fault event
  OB82_FLT_ID : BYTE ;	//16#XX, Fault identifcation code
  OB82_PRIORITY : BYTE ;	//Priority of OB Execution
  OB82_OB_NUMBR : BYTE ;	//82 (Organization block 82, OB82)
  OB82_RESERVED_1 : BYTE ;	//Reserved for system
  OB82_IO_FLAG : BYTE ;	//Input (01010100), Output (01010101)
  OB82_MDL_ADDR : WORD ;	//Base address of module with fault
  OB82_MDL_DEFECT : BOOL ;	//Module defective
  OB82_INT_FAULT : BOOL ;	//Internal fault
  OB82_EXT_FAULT : BOOL ;	//External fault
  OB82_PNT_INFO : BOOL ;	//Point information
  OB82_EXT_VOLTAGE : BOOL ;	//External voltage low
  OB82_FLD_CONNCTR : BOOL ;	//Field wiring connector missing
  OB82_NO_CONFIG : BOOL ;	//Module has no configuration data
  OB82_CONFIG_ERR : BOOL ;	//Module has configuration error
  OB82_MDL_TYPE : BYTE ;	//Type of module
  OB82_SUB_MDL_ERR : BOOL ;	//Sub-Module is missing or has error
  OB82_COMM_FAULT : BOOL ;	//Communication fault
  OB82_MDL_STOP : BOOL ;	//Module is stopped
  OB82_WTCH_DOG_FLT : BOOL ;	//Watch dog timer stopped module
  OB82_INT_PS_FLT : BOOL ;	//Internal power supply fault
  OB82_PRIM_BATT_FLT : BOOL ;	//Primary battery is in fault
  OB82_BCKUP_BATT_FLT : BOOL ;	//Backup battery is in fault
  OB82_RESERVED_2 : BOOL ;	//Reserved for system
  OB82_RACK_FLT : BOOL ;	//Rack fault, only for bus interface module
  OB82_PROC_FLT : BOOL ;	//Processor fault
  OB82_EPROM_FLT : BOOL ;	//EPROM fault
  OB82_RAM_FLT : BOOL ;	//RAM fault
  OB82_ADU_FLT : BOOL ;	//ADU fault
  OB82_FUSE_FLT : BOOL ;	//Fuse fault
  OB82_HW_INTR_FLT : BOOL ;	//Hardware interupt input in fault
  OB82_RESERVED_3 : BOOL ;	//Reserved for system
  OB82_DATE_TIME : DATE_AND_TIME ;	//Date and time OB82 started
END_VAR
BEGIN
NETWORK
TITLE = Detailed Diagnosis in OB82 (interrupt)
      CALL  "GP_DIAG" (
           $1                       := TRUE);
END_ORGANIZATION_BLOCK

ORGANIZATION_BLOCK OB 86
TITLE = "Loss Of Rack Fault"
VERSION : 1.0
VAR_TEMP
  OB86_EV_CLASS : BYTE ;	//16#38/39 Event class 3
  OB86_FLT_ID : BYTE ;	//16#C1/C4/C5, Fault identifcation code
  OB86_PRIORITY : BYTE ;	//Priority of OB Execution
  OB86_OB_NUMBR : BYTE ;	//86 (Organization block 86, OB86)
  OB86_RESERVED_1 : BYTE ;	//Reserved for system
  OB86_RESERVED_2 : BYTE ;	//Reserved for system
  OB86_MDL_ADDR : WORD ;	//Base address of IM module in rack with fault
  OB86_RACKS_FLTD : ARRAY  [0 .. 31 ] OF BOOL ;	//Racks in fault
  OB86_DATE_TIME : DATE_AND_TIME ;	//Date and time OB86 started
END_VAR
BEGIN
NETWORK
TITLE = Detailed Diagnosis in OB86 (interrupt)
      CALL  "GP_DIAG" (
           $1                       := TRUE);
END_ORGANIZATION_BLOCK

ORGANIZATION_BLOCK "COMPLETE RESTART"	// OB 100
TITLE = "Complete Restart"
VERSION : 0.1
VAR_TEMP
  OB100_EV_CLASS : BYTE ;	//16#13, Event class 1, Entering event state, Event logged in diagnostic buffer
  OB100_STRTUP : BYTE ;	//16#81/82/83/84 Method of startup
  OB100_PRIORITY : BYTE ;	//Priority of OB Execution
  OB100_OB_NUMBR : BYTE ;	//100 (Organization block 100, OB100)
  OB100_RESERVED_1 : BYTE ;	//Reserved for system
  OB100_RESERVED_2 : BYTE ;	//Reserved for system
  OB100_STOP : WORD ;	//Event that caused CPU to stop (16#4xxx)
  OB100_STRT_INFO : DWORD ;	//Information on how system started
  OB100_DATE_TIME : DATE_AND_TIME ;	//Date and time OB100 started
END_VAR
BEGIN
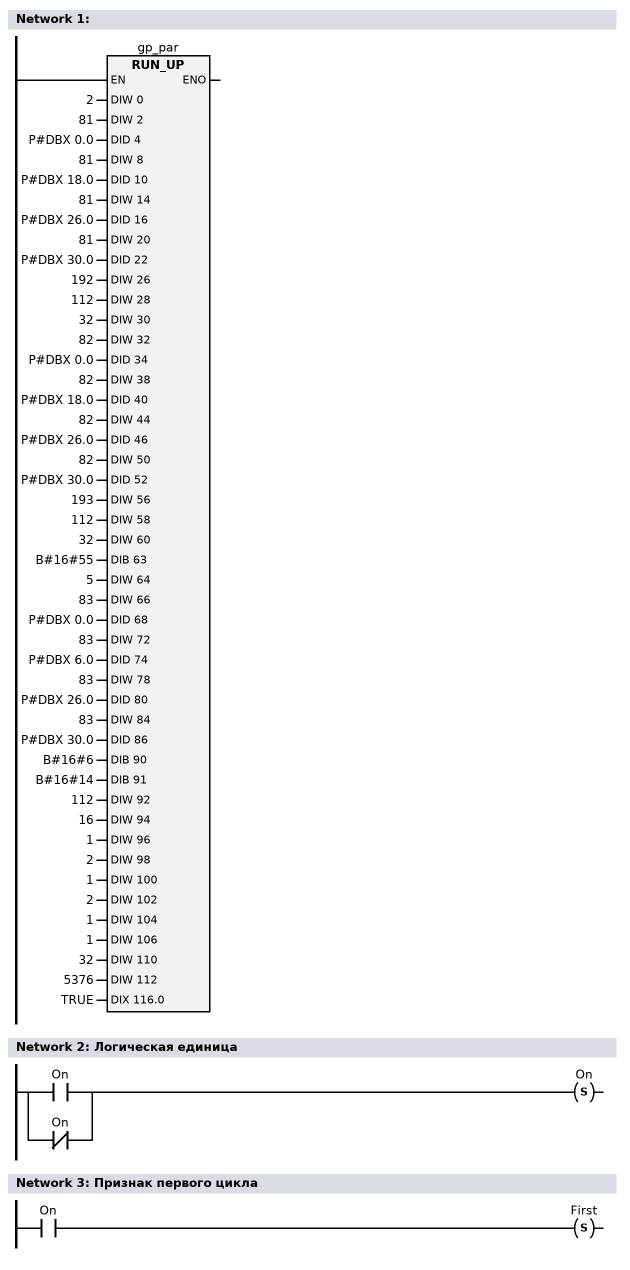
NETWORK
TITLE =
      CALL  "RUN_UP" , "gp_par" (
           DIW 0                    := 2,
           DIW 2                    := 81,
           DID 4                    := P#DBX 0.0,
           DIW 8                    := 81,
           DID 10                   := P#DBX 18.0,
           DIW 14                   := 81,
           DID 16                   := P#DBX 26.0,
           DIW 20                   := 81,
           DID 22                   := P#DBX 30.0,
           DIW 26                   := 192,
           DIW 28                   := 112,
           DIW 30                   := 32,
           DIW 32                   := 82,
           DID 34                   := P#DBX 0.0,
           DIW 38                   := 82,
           DID 40                   := P#DBX 18.0,
           DIW 44                   := 82,
           DID 46                   := P#DBX 26.0,
           DIW 50                   := 82,
           DID 52                   := P#DBX 30.0,
           DIW 56                   := 193,
           DIW 58                   := 112,
           DIW 60                   := 32,
           DIB 63                   := B#16#55,
           DIW 64                   := 5,
           DIW 66                   := 83,
           DID 68                   := P#DBX 0.0,
           DIW 72                   := 83,
           DID 74                   := P#DBX 6.0,
           DIW 78                   := 83,
           DID 80                   := P#DBX 26.0,
           DIW 84                   := 83,
           DID 86                   := P#DBX 30.0,
           DIB 90                   := B#16#6,
           DIB 91                   := B#16#14,
           DIW 92                   := 112,
           DIW 94                   := 16,
           DIW 96                   := 1,
           DIW 98                   := 2,
           DIW 100                  := 1,
           DIW 102                  := 2,
           DIW 104                  := 1,
           DIW 106                  := 1,
           DIW 110                  := 32,
           DIW 112                  := 5376,
           DIX 116.0                := TRUE);
NETWORK
TITLE = Логическая единица
      O     "On";
      ON    "On";
      S     "On";
NETWORK
TITLE = Признак первого цикла
      A     "On";
      S     "First";
END_ORGANIZATION_BLOCK
